Yaskawa INFORM job: DEMO_ROOF_SIDE_0625_3PAINT_38.JBI

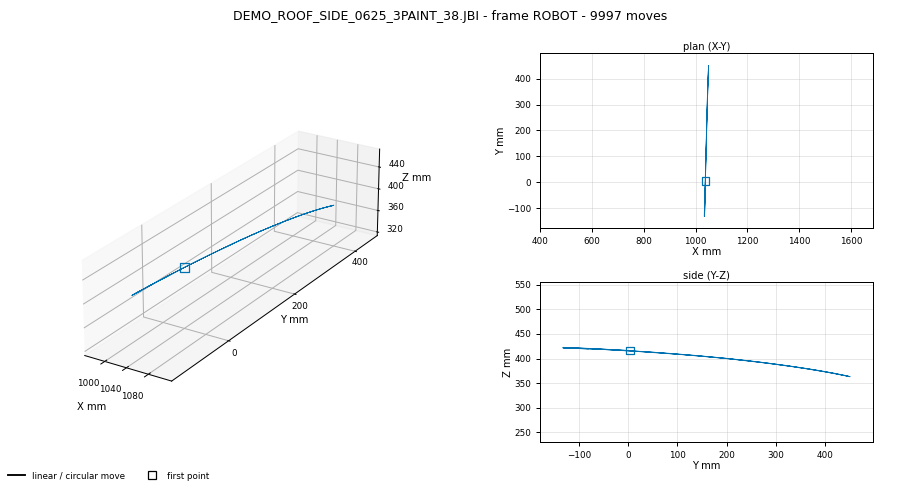
[picture p0: tool path of DEMO_ROOF_SIDE_0625_3PAINT_38.JBI in frame ROBOT, 9997 of 9997 moves have a stored position in this frame; points joined in program order, loops and branches not executed]
/JOB
//NAME DEMO_ROOF_SIDE_0625_3PAINT38
//POS
///NPOS 9997,0,0,0,0,0
///TOOL 0
///USER 0
///POSTYPE ROBOT
///RECTAN
///RCONF 1,0,0,0,0,0,0,0,0,0,0,0,0,0,0,0,0,0,0,0,0,0,0,0
C00000=1038.595,4.241,416.318,169.157,38.319,157.198
C00001=1038.590,3.992,416.332,169.155,38.320,157.198
C00002=1038.583,3.742,416.347,169.153,38.319,157.198
C00003=1038.577,3.493,416.362,169.151,38.318,157.198
C00004=1038.570,3.243,416.378,169.149,38.318,157.198
C00005=1038.564,2.994,416.393,169.147,38.318,157.198
C00006=1038.557,2.744,416.408,169.145,38.317,157.197
C00007=1038.552,2.495,416.422,169.142,38.317,157.197
C00008=1038.545,2.246,416.437,169.140,38.317,157.197
C00009=1038.539,1.996,416.452,169.138,38.316,157.197
C00010=1038.532,1.746,416.467,169.136,38.316,157.197
C00011=1038.526,1.497,416.482,169.134,38.315,157.197
C00012=1038.519,1.248,416.498,169.132,38.315,157.197
C00013=1038.514,0.999,416.513,169.130,38.315,157.197
C00014=1038.507,0.749,416.527,169.128,38.314,157.197
C00015=1038.501,0.499,416.542,169.125,38.314,157.196
C00016=1038.495,0.249,416.558,169.123,38.314,157.196
C00017=1038.489,-0.000,416.573,169.121,38.313,157.196
C00018=1038.483,-0.249,416.587,169.119,38.313,157.196
C00019=1038.477,-0.499,416.602,169.116,38.313,157.196
C00020=1038.470,-0.749,416.617,169.114,38.312,157.196
C00021=1038.464,-0.998,416.632,169.112,38.312,157.196
C00022=1038.458,-1.247,416.647,169.110,38.311,157.196
C00023=1038.452,-1.497,416.662,169.108,38.311,157.196
C00024=1038.445,-1.747,416.677,169.106,38.311,157.196
C00025=1038.439,-1.996,416.692,169.104,38.310,157.195
C00026=1038.433,-2.245,416.706,169.102,38.310,157.195
C00027=1038.427,-2.495,416.721,169.100,38.310,157.195
C00028=1038.420,-2.744,416.736,169.098,38.309,157.195
C00029=1038.414,-2.994,416.751,169.096,38.309,157.195
C00030=1038.407,-3.278,416.767,169.092,38.308,157.195
C00031=1038.400,-3.560,416.785,169.090,38.308,157.195
C00032=1038.393,-3.844,416.802,169.087,38.308,157.195
C00033=1038.385,-4.127,416.817,169.085,38.307,157.194
C00034=1038.379,-4.377,416.832,169.083,38.307,157.194
C00035=1038.373,-4.627,416.847,169.081,38.307,157.194
C00036=1038.366,-4.876,416.862,169.079,38.307,157.194
C00037=1038.360,-5.125,416.876,169.076,38.306,157.194
C00038=1038.354,-5.375,416.890,169.074,38.306,157.194
C00039=1038.347,-5.625,416.905,169.072,38.306,157.194
C00040=1038.340,-5.874,416.920,169.070,38.306,157.194
C00041=1038.334,-6.123,416.934,169.068,38.305,157.194
C00042=1038.328,-6.373,416.949,169.066,38.306,157.194
C00043=1038.321,-6.623,416.963,169.064,38.305,157.194
C00044=1038.315,-6.873,416.978,169.061,38.304,157.193
C00045=1038.309,-7.122,416.992,169.058,38.305,157.193
C00046=1038.303,-7.371,417.007,169.056,38.304,157.193
C00047=1038.296,-7.621,417.021,169.054,38.304,157.193
C00048=1038.290,-7.870,417.035,169.052,38.304,157.193
C00049=1038.284,-8.120,417.050,169.050,38.304,157.193
C00050=1038.277,-8.369,417.065,169.048,38.303,157.193
C00051=1038.271,-8.619,417.079,169.046,38.303,157.193
C00052=1038.265,-8.868,417.094,169.043,38.303,157.193
C00053=1038.258,-9.118,417.108,169.041,38.303,157.193
C00054=1038.252,-9.367,417.123,169.039,38.302,157.193
C00055=1038.246,-9.617,417.137,169.037,38.302,157.192
C00056=1038.239,-9.866,417.151,169.035,38.302,157.192
C00057=1038.233,-10.115,417.166,169.033,38.301,157.192
C00058=1038.227,-10.365,417.180,169.030,38.301,157.192
C00059=1038.220,-10.615,417.194,169.027,38.301,157.192
C00060=1038.214,-10.864,417.209,169.025,38.301,157.192
C00061=1038.208,-11.114,417.223,169.023,38.300,157.192
C00062=1038.201,-11.363,417.237,169.021,38.300,157.192
C00063=1038.195,-11.613,417.251,169.019,38.300,157.192
C00064=1038.189,-11.863,417.266,169.017,38.299,157.192
C00065=1038.182,-12.111,417.280,169.015,38.299,157.192
C00066=1038.176,-12.362,417.294,169.012,38.299,157.191
C00067=1038.170,-12.611,417.309,169.010,38.299,157.191
C00068=1038.163,-12.860,417.323,169.008,38.298,157.191
C00069=1038.157,-13.110,417.338,169.006,38.299,157.191
C00070=1038.151,-13.359,417.352,169.004,38.298,157.191
C00071=1038.145,-13.609,417.366,169.002,38.298,157.191
C00072=1038.139,-13.858,417.380,168.998,38.298,157.191
C00073=1038.132,-14.108,417.394,168.996,38.298,157.191
C00074=1038.126,-14.358,417.409,168.994,38.297,157.191
C00075=1038.120,-14.607,417.423,168.992,38.297,157.191
C00076=1038.113,-14.857,417.437,168.990,38.297,157.191
C00077=1038.107,-15.105,417.452,168.988,38.296,157.190
C00078=1038.101,-15.356,417.466,168.985,38.296,157.190
C00079=1038.095,-15.605,417.479,168.983,38.296,157.190
C00080=1038.088,-15.854,417.494,168.981,38.296,157.190
C00081=1038.082,-16.105,417.508,168.979,38.296,157.190
C00082=1038.075,-16.353,417.522,168.977,38.295,157.190
C00083=1038.069,-16.604,417.536,168.974,38.295,157.190
C00084=1038.063,-16.852,417.550,168.972,38.295,157.190
C00085=1038.056,-17.102,417.564,168.970,38.295,157.190
C00086=1038.050,-17.352,417.578,168.968,38.294,157.190
C00087=1038.043,-17.601,417.592,168.966,38.295,157.190
C00088=1038.037,-17.851,417.606,168.963,38.295,157.190
C00089=1038.031,-18.100,417.620,168.960,38.294,157.190
C00090=1038.024,-18.350,417.634,168.958,38.294,157.190
C00091=1038.018,-18.600,417.648,168.956,38.294,157.189
C00092=1038.011,-18.849,417.662,168.954,38.294,157.189
C00093=1038.005,-19.098,417.675,168.951,38.294,157.189
C00094=1037.998,-19.380,417.692,168.949,38.293,157.189
C00095=1037.992,-19.662,417.707,168.946,38.293,157.189
C00096=1037.984,-19.944,417.723,168.944,38.293,157.189
C00097=1037.977,-20.226,417.738,168.941,38.293,157.189
C00098=1037.970,-20.475,417.752,168.939,38.292,157.189
C00099=1037.964,-20.725,417.766,168.937,38.293,157.189
C00100=1037.958,-20.975,417.780,168.935,38.293,157.189
C00101=1037.951,-21.224,417.794,168.932,38.292,157.189
C00102=1037.945,-21.473,417.808,168.930,38.292,157.189
C00103=1037.939,-21.723,417.822,168.928,38.292,157.188
C00104=1037.932,-21.973,417.835,168.926,38.292,157.188
C00105=1037.926,-22.223,417.849,168.923,38.291,157.188
C00106=1037.920,-22.472,417.863,168.920,38.291,157.188
C00107=1037.914,-22.721,417.877,168.918,38.291,157.188
C00108=1037.908,-22.971,417.891,168.916,38.291,157.188
C00109=1037.901,-23.220,417.904,168.914,38.291,157.188
C00110=1037.894,-23.470,417.918,168.911,38.290,157.188
C00111=1037.889,-23.719,417.932,168.909,38.291,157.188
C00112=1037.882,-23.969,417.946,168.907,38.291,157.188
C00113=1037.876,-24.219,417.959,168.905,38.290,157.188
C00114=1037.870,-24.468,417.973,168.903,38.290,157.188
C00115=1037.863,-24.717,417.987,168.900,38.290,157.188
C00116=1037.857,-24.967,418.001,168.898,38.290,157.188
C00117=1037.851,-25.217,418.015,168.896,38.290,157.188
C00118=1037.845,-25.466,418.028,168.894,38.289,157.187
C00119=1037.838,-25.716,418.041,168.891,38.289,157.187
C00120=1037.832,-25.966,418.056,168.889,38.289,157.187
C00121=1037.826,-26.215,418.069,168.887,38.289,157.187
C00122=1037.820,-26.464,418.082,168.885,38.288,157.187
C00123=1037.813,-26.714,418.097,168.881,38.289,157.187
C00124=1037.807,-26.963,418.110,168.879,38.289,157.187
C00125=1037.800,-27.213,418.124,168.877,38.288,157.187
C00126=1037.794,-27.462,418.137,168.875,38.288,157.187
C00127=1037.789,-27.712,418.151,168.872,38.288,157.187
C00128=1037.782,-27.962,418.165,168.870,38.288,157.187
C00129=1037.776,-28.211,418.178,168.868,38.288,157.187
C00130=1037.769,-28.461,418.191,168.865,38.288,157.187
C00131=1037.763,-28.711,418.205,168.863,38.288,157.187
C00132=1037.756,-28.960,418.218,168.861,38.288,157.187
C00133=1037.750,-29.210,418.232,168.859,38.288,157.186
C00134=1037.743,-29.459,418.245,168.856,38.288,157.186
C00135=1037.737,-29.708,418.258,168.854,38.288,157.186
C00136=1037.731,-29.959,418.271,168.852,38.287,157.186
C00137=1037.725,-30.208,418.285,168.849,38.287,157.186
C00138=1037.718,-30.457,418.298,168.847,38.288,157.186
C00139=1037.712,-30.708,418.312,168.845,38.288,157.186
C00140=1037.706,-30.957,418.325,168.843,38.287,157.186
C00141=1037.700,-31.206,418.339,168.840,38.287,157.186
C00142=1037.693,-31.456,418.352,168.838,38.287,157.186
C00143=1037.687,-31.705,418.366,168.836,38.287,157.186
C00144=1037.681,-31.955,418.379,168.833,38.287,157.186
C00145=1037.674,-32.204,418.392,168.831,38.287,157.186
C00146=1037.668,-32.455,418.405,168.829,38.287,157.186
C00147=1037.662,-32.704,418.418,168.826,38.287,157.186
C00148=1037.655,-32.953,418.432,168.823,38.287,157.185
C00149=1037.649,-33.203,418.445,168.821,38.287,157.185
C00150=1037.642,-33.452,418.458,168.819,38.287,157.185
C00151=1037.636,-33.702,418.472,168.816,38.287,157.185
C00152=1037.630,-33.951,418.485,168.814,38.286,157.185
C00153=1037.623,-34.201,418.498,168.812,38.287,157.185
C00154=1037.617,-34.451,418.511,168.809,38.287,157.185
C00155=1037.611,-34.700,418.524,168.807,38.287,157.185
C00156=1037.605,-34.949,418.538,168.805,38.286,157.185
C00157=1037.598,-35.200,418.551,168.802,38.286,157.185
C00158=1037.592,-35.480,418.566,168.800,38.286,157.185
C00159=1037.585,-35.762,418.580,168.797,38.287,157.185
C00160=1037.578,-36.043,418.596,168.795,38.286,157.185
C00161=1037.571,-36.323,418.610,168.792,38.286,157.185
C00162=1037.564,-36.573,418.624,168.790,38.286,157.185
C00163=1037.558,-36.823,418.637,168.787,38.286,157.185
C00164=1037.552,-37.073,418.650,168.785,38.286,157.185
C00165=1037.546,-37.322,418.663,168.783,38.286,157.185
C00166=1037.540,-37.571,418.676,168.780,38.286,157.184
C00167=1037.533,-37.822,418.689,168.778,38.286,157.184
C00168=1037.527,-38.071,418.702,168.776,38.286,157.184
C00169=1037.521,-38.320,418.716,168.773,38.286,157.184
C00170=1037.515,-38.570,418.728,168.771,38.286,157.184
C00171=1037.508,-38.819,418.742,168.769,38.286,157.184
C00172=1037.502,-39.069,418.755,168.766,38.286,157.184
C00173=1037.496,-39.319,418.768,168.763,38.286,157.184
C00174=1037.490,-39.568,418.781,168.761,38.286,157.184
C00175=1037.483,-39.818,418.793,168.758,38.286,157.184
C00176=1037.477,-40.067,418.806,168.756,38.286,157.184
C00177=1037.470,-40.317,418.820,168.754,38.286,157.184
C00178=1037.465,-40.566,418.832,168.751,38.286,157.184
C00179=1037.458,-40.816,418.846,168.749,38.286,157.184
C00180=1037.451,-41.066,418.858,168.746,38.286,157.184
C00181=1037.445,-41.315,418.871,168.744,38.286,157.184
C00182=1037.439,-41.565,418.883,168.742,38.286,157.184
C00183=1037.433,-41.814,418.897,168.739,38.287,157.184
C00184=1037.426,-42.064,418.909,168.737,38.286,157.184
C00185=1037.420,-42.313,418.922,168.735,38.286,157.184
C00186=1037.413,-42.564,418.935,168.732,38.286,157.184
C00187=1037.407,-42.813,418.948,168.730,38.286,157.184
C00188=1037.401,-43.063,418.960,168.727,38.287,157.184
C00189=1037.394,-43.312,418.973,168.725,38.287,157.184
C00190=1037.388,-43.562,418.986,168.723,38.287,157.183
C00191=1037.382,-43.811,418.999,168.720,38.287,157.183
C00192=1037.376,-44.061,419.012,168.718,38.287,157.183
C00193=1037.370,-44.310,419.024,168.716,38.287,157.183
C00194=1037.363,-44.560,419.037,168.713,38.287,157.183
C00195=1037.358,-44.810,419.050,168.711,38.287,157.183
C00196=1037.351,-45.059,419.063,168.708,38.287,157.183
C00197=1037.345,-45.308,419.075,168.706,38.287,157.183
C00198=1037.338,-45.559,419.088,168.704,38.287,157.183
C00199=1037.332,-45.808,419.101,168.701,38.287,157.183
C00200=1037.325,-46.058,419.113,168.699,38.287,157.183
C00201=1037.319,-46.307,419.126,168.696,38.287,157.183
C00202=1037.313,-46.557,419.139,168.694,38.287,157.183
C00203=1037.307,-46.807,419.151,168.692,38.288,157.183
C00204=1037.300,-47.056,419.164,168.689,38.288,157.183
C00205=1037.294,-47.306,419.177,168.687,38.288,157.183
C00206=1037.288,-47.556,419.189,168.684,38.288,157.183
C00207=1037.282,-47.805,419.202,168.682,38.288,157.183
C00208=1037.276,-48.054,419.214,168.680,38.288,157.183
C00209=1037.270,-48.304,419.227,168.677,38.288,157.183
C00210=1037.264,-48.554,419.239,168.675,38.288,157.183
C00211=1037.257,-48.803,419.252,168.673,38.288,157.183
C00212=1037.251,-49.053,419.265,168.670,38.288,157.183
C00213=1037.245,-49.303,419.277,168.668,38.288,157.183
C00214=1037.239,-49.552,419.290,168.665,38.288,157.183
C00215=1037.232,-49.802,419.302,168.663,38.288,157.183
C00216=1037.227,-50.051,419.315,168.659,38.288,157.183
C00217=1037.221,-50.301,419.327,168.657,38.288,157.182
C00218=1037.214,-50.550,419.339,168.655,38.289,157.182
C00219=1037.208,-50.800,419.352,168.652,38.289,157.182
C00220=1037.201,-51.049,419.364,168.650,38.289,157.182
C00221=1037.196,-51.299,419.377,168.648,38.290,157.182
C00222=1037.188,-51.581,419.390,168.646,38.290,157.182
C00223=1037.180,-51.862,419.404,168.642,38.290,157.182
C00224=1037.173,-52.144,419.418,168.639,38.290,157.182
C00225=1037.166,-52.426,419.433,168.636,38.290,157.182
C00226=1037.160,-52.675,419.444,168.635,38.291,157.182
C00227=1037.153,-52.924,419.456,168.632,38.291,157.182
C00228=1037.147,-53.174,419.469,168.630,38.291,157.182
C00229=1037.141,-53.424,419.481,168.626,38.291,157.182
C00230=1037.134,-53.673,419.493,168.624,38.291,157.182
C00231=1037.128,-53.923,419.505,168.621,38.291,157.182
C00232=1037.122,-54.173,419.517,168.620,38.292,157.182
C00233=1037.115,-54.422,419.529,168.617,38.292,157.182
C00234=1037.109,-54.672,419.542,168.615,38.292,157.182
C00235=1037.102,-54.922,419.554,168.612,38.293,157.182
C00236=1037.096,-55.172,419.566,168.609,38.293,157.182
C00237=1037.090,-55.421,419.578,168.607,38.293,157.182
C00238=1037.083,-55.671,419.590,168.605,38.294,157.182
C00239=1037.077,-55.921,419.603,168.602,38.294,157.182
C00240=1037.071,-56.170,419.615,168.600,38.294,157.182
C00241=1037.065,-56.419,419.626,168.597,38.294,157.182
C00242=1037.059,-56.669,419.639,168.595,38.295,157.182
C00243=1037.052,-56.919,419.651,168.592,38.295,157.182
C00244=1037.045,-57.168,419.663,168.590,38.295,157.182
C00245=1037.039,-57.418,419.675,168.588,38.295,157.182
C00246=1037.033,-57.668,419.687,168.585,38.295,157.182
C00247=1037.026,-57.918,419.698,168.583,38.296,157.182
C00248=1037.020,-58.167,419.710,168.580,38.296,157.182
C00249=1037.014,-58.416,419.723,168.578,38.296,157.182
C00250=1037.008,-58.666,419.735,168.575,38.296,157.182
C00251=1037.001,-58.916,419.746,168.573,38.296,157.182
C00252=1036.995,-59.166,419.759,168.570,38.297,157.182
C00253=1036.989,-59.415,419.771,168.568,38.297,157.182
C00254=1036.983,-59.664,419.783,168.565,38.297,157.182
C00255=1036.977,-59.914,419.794,168.563,38.297,157.182
C00256=1036.970,-60.164,419.806,168.560,38.298,157.182
C00257=1036.964,-60.414,419.818,168.558,38.298,157.182
C00258=1036.958,-60.663,419.831,168.555,38.298,157.182
C00259=1036.952,-60.912,419.843,168.553,38.299,157.182
C00260=1036.945,-61.163,419.854,168.550,38.299,157.182
C00261=1036.939,-61.412,419.866,168.548,38.299,157.182
C00262=1036.933,-61.662,419.878,168.545,38.300,157.182
C00263=1036.926,-61.912,419.890,168.543,38.300,157.182
C00264=1036.920,-62.160,419.902,168.540,38.300,157.182
C00265=1036.915,-62.411,419.914,168.538,38.300,157.182
C00266=1036.908,-62.661,419.926,168.535,38.301,157.182
C00267=1036.901,-62.910,419.938,168.533,38.301,157.182
C00268=1036.895,-63.159,419.949,168.530,38.301,157.182
C00269=1036.890,-63.409,419.961,168.527,38.301,157.182
C00270=1036.883,-63.659,419.973,168.525,38.302,157.182
C00271=1036.877,-63.908,419.985,168.522,38.302,157.182
C00272=1036.871,-64.158,419.996,168.520,38.302,157.182
C00273=1036.865,-64.408,420.008,168.517,38.302,157.182
C00274=1036.858,-64.658,420.020,168.515,38.303,157.182
C00275=1036.852,-64.907,420.031,168.512,38.303,157.182
C00276=1036.846,-65.157,420.044,168.510,38.303,157.182
C00277=1036.840,-65.407,420.056,168.507,38.303,157.182
C00278=1036.834,-65.656,420.067,168.505,38.303,157.182
C00279=1036.827,-65.906,420.079,168.502,38.304,157.182
C00280=1036.821,-66.155,420.091,168.500,38.304,157.182
C00281=1036.816,-66.405,420.102,168.497,38.304,157.182
C00282=1036.809,-66.655,420.114,168.495,38.305,157.182
C00283=1036.802,-66.904,420.126,168.492,38.305,157.182
C00284=1036.797,-67.154,420.137,168.490,38.305,157.182
C00285=1036.791,-67.403,420.149,168.487,38.306,157.182
C00286=1036.784,-67.686,420.162,168.484,38.306,157.182
C00287=1036.777,-67.969,420.175,168.481,38.307,157.182
C00288=1036.770,-68.252,420.189,168.479,38.307,157.182
C00289=1036.763,-68.535,420.202,168.476,38.307,157.182
C00290=1036.757,-68.784,420.214,168.473,38.308,157.182
C00291=1036.751,-69.034,420.225,168.471,38.308,157.182
C00292=1036.745,-69.284,420.237,168.468,38.308,157.182
C00293=1036.739,-69.533,420.248,168.466,38.308,157.182
C00294=1036.733,-69.783,420.260,168.463,38.309,157.182
C00295=1036.726,-70.033,420.271,168.461,38.309,157.182
C00296=1036.720,-70.282,420.283,168.458,38.309,157.182
C00297=1036.715,-70.532,420.295,168.455,38.309,157.182
C00298=1036.708,-70.781,420.306,168.453,38.310,157.182
C00299=1036.702,-71.032,420.317,168.450,38.310,157.182
C00300=1036.696,-71.280,420.329,168.448,38.310,157.182
C00301=1036.690,-71.531,420.341,168.445,38.311,157.182
C00302=1036.684,-71.780,420.352,168.443,38.311,157.182
C00303=1036.678,-72.030,420.364,168.440,38.311,157.182
C00304=1036.672,-72.279,420.375,168.438,38.311,157.182
C00305=1036.666,-72.529,420.387,168.435,38.312,157.182
C00306=1036.661,-72.779,420.398,168.433,38.312,157.182
C00307=1036.654,-73.028,420.410,168.430,38.312,157.182
C00308=1036.648,-73.278,420.421,168.428,38.312,157.182
C00309=1036.642,-73.528,420.432,168.425,38.313,157.182
C00310=1036.635,-73.778,420.444,168.422,38.313,157.182
C00311=1036.630,-74.027,420.455,168.420,38.313,157.182
C00312=1036.624,-74.278,420.467,168.417,38.314,157.182
C00313=1036.617,-74.526,420.478,168.415,38.314,157.182
C00314=1036.611,-74.776,420.489,168.412,38.315,157.182
C00315=1036.605,-75.026,420.500,168.410,38.315,157.182
C00316=1036.598,-75.275,420.512,168.407,38.316,157.182
C00317=1036.593,-75.525,420.523,168.404,38.316,157.182
C00318=1036.586,-75.775,420.534,168.402,38.317,157.182
C00319=1036.581,-76.025,420.545,168.399,38.317,157.182
C00320=1036.574,-76.274,420.557,168.397,38.318,157.182
C00321=1036.568,-76.524,420.568,168.394,38.318,157.182
C00322=1036.562,-76.774,420.579,168.392,38.319,157.182
C00323=1036.556,-77.023,420.590,168.390,38.319,157.182
C00324=1036.550,-77.274,420.601,168.387,38.320,157.182
C00325=1036.544,-77.522,420.613,168.385,38.320,157.182
C00326=1036.537,-77.773,420.624,168.382,38.320,157.183
C00327=1036.531,-78.022,420.634,168.379,38.321,157.182
C00328=1036.525,-78.271,420.645,168.377,38.321,157.183
C00329=1036.519,-78.521,420.656,168.374,38.321,157.183
C00330=1036.513,-78.771,420.667,168.372,38.322,157.183
C00331=1036.507,-79.021,420.679,168.369,38.322,157.183
C00332=1036.501,-79.270,420.690,168.366,38.323,157.183
C00333=1036.494,-79.520,420.701,168.364,38.323,157.183
C00334=1036.489,-79.770,420.712,168.361,38.324,157.183
C00335=1036.483,-80.019,420.723,168.359,38.324,157.183
C00336=1036.476,-80.269,420.734,168.356,38.325,157.183
C00337=1036.470,-80.519,420.744,168.353,38.325,157.183
C00338=1036.464,-80.769,420.756,168.351,38.326,157.183
C00339=1036.457,-81.018,420.766,168.348,38.327,157.183
C00340=1036.451,-81.268,420.777,168.345,38.327,157.183
C00341=1036.445,-81.518,420.788,168.343,38.328,157.183
C00342=1036.438,-81.767,420.799,168.340,38.328,157.183
C00343=1036.432,-82.017,420.810,168.337,38.329,157.183
C00344=1036.427,-82.266,420.821,168.335,38.329,157.183
C00345=1036.420,-82.516,420.831,168.333,38.330,157.183
C00346=1036.414,-82.766,420.842,168.330,38.331,157.183
C00347=1036.408,-83.016,420.853,168.328,38.331,157.183
C00348=1036.401,-83.265,420.864,168.325,38.332,157.183
C00349=1036.395,-83.515,420.874,168.322,38.333,157.183
C00350=1036.388,-83.800,420.887,168.319,38.333,157.183
C00351=1036.381,-84.085,420.899,168.316,38.334,157.183
C00352=1036.374,-84.370,420.911,168.313,38.334,157.184
C00353=1036.367,-84.655,420.923,168.310,38.335,157.184
C00354=1036.361,-84.905,420.934,168.308,38.336,157.184
C00355=1036.354,-85.154,420.944,168.305,38.336,157.184
C00356=1036.349,-85.404,420.955,168.302,38.337,157.184
C00357=1036.342,-85.654,420.967,168.300,38.338,157.184
C00358=1036.336,-85.903,420.977,168.297,38.338,157.184
C00359=1036.330,-86.152,420.988,168.294,38.339,157.184
C00360=1036.323,-86.402,420.998,168.292,38.339,157.184
C00361=1036.318,-86.652,421.009,168.289,38.340,157.184
C00362=1036.312,-86.902,421.019,168.286,38.340,157.184
C00363=1036.305,-87.152,421.030,168.285,38.341,157.184
C00364=1036.299,-87.401,421.041,168.282,38.342,157.184
C00365=1036.293,-87.651,421.052,168.279,38.343,157.184
C00366=1036.287,-87.901,421.061,168.277,38.343,157.184
C00367=1036.281,-88.151,421.073,168.274,38.343,157.184
C00368=1036.274,-88.400,421.083,168.271,38.344,157.184
C00369=1036.269,-88.649,421.094,168.268,38.345,157.184
C00370=1036.263,-88.900,421.104,168.266,38.345,157.184
C00371=1036.256,-89.149,421.115,168.263,38.346,157.185
C00372=1036.250,-89.399,421.126,168.260,38.347,157.185
C00373=1036.244,-89.648,421.136,168.258,38.348,157.185
C00374=1036.238,-89.899,421.146,168.255,38.348,157.185
C00375=1036.232,-90.148,421.157,168.252,38.349,157.185
C00376=1036.226,-90.398,421.167,168.250,38.349,157.185
C00377=1036.220,-90.648,421.178,168.247,38.350,157.185
C00378=1036.214,-90.897,421.188,168.244,38.350,157.185
C00379=1036.207,-91.147,421.199,168.242,38.351,157.185
C00380=1036.201,-91.396,421.209,168.240,38.352,157.185
C00381=1036.195,-91.646,421.220,168.237,38.353,157.185
C00382=1036.190,-91.896,421.230,168.235,38.353,157.185
C00383=1036.184,-92.146,421.240,168.232,38.353,157.185
C00384=1036.178,-92.395,421.251,168.229,38.354,157.185
C00385=1036.171,-92.645,421.262,168.227,38.355,157.185
C00386=1036.165,-92.895,421.272,168.224,38.355,157.185
C00387=1036.160,-93.145,421.283,168.221,38.356,157.185
C00388=1036.153,-93.394,421.293,168.219,38.357,157.185
C00389=1036.148,-93.644,421.303,168.216,38.358,157.186
C00390=1036.141,-93.893,421.313,168.213,38.358,157.186
C00391=1036.135,-94.144,421.324,168.211,38.358,157.186
C00392=1036.129,-94.393,421.334,168.208,38.359,157.186
C00393=1036.123,-94.643,421.344,168.205,38.360,157.186
C00394=1036.117,-94.892,421.355,168.202,38.361,157.186
C00395=1036.111,-95.142,421.365,168.200,38.361,157.186
C00396=1036.106,-95.392,421.376,168.197,38.362,157.186
C00397=1036.099,-95.641,421.386,168.195,38.363,157.186
C00398=1036.094,-95.891,421.396,168.193,38.363,157.186
C00399=1036.087,-96.140,421.406,168.190,38.364,157.186
C00400=1036.082,-96.390,421.417,168.187,38.364,157.186
C00401=1036.075,-96.640,421.427,168.185,38.365,157.186
C00402=1036.069,-96.890,421.437,168.182,38.366,157.186
C00403=1036.063,-97.140,421.448,168.179,38.367,157.186
C00404=1036.057,-97.390,421.458,168.177,38.367,157.186
C00405=1036.051,-97.640,421.467,168.174,38.368,157.187
C00406=1036.045,-97.889,421.478,168.171,38.369,157.187
C00407=1036.039,-98.139,421.488,168.168,38.370,157.187
C00408=1036.033,-98.388,421.498,168.166,38.371,157.187
C00409=1036.027,-98.638,421.508,168.163,38.371,157.187
C00410=1036.021,-98.888,421.518,168.161,38.372,157.187
C00411=1036.015,-99.137,421.528,168.158,38.373,157.187
C00412=1036.008,-99.387,421.538,168.156,38.374,157.187
C00413=1036.002,-99.638,421.548,168.153,38.375,157.187
C00414=1035.993,-100.042,421.564,168.148,38.376,157.187
C00415=1035.983,-100.445,421.581,168.144,38.377,157.187
C00416=1035.972,-100.849,421.597,168.140,38.378,157.187
C00417=1035.963,-101.253,421.613,168.135,38.379,157.188
C00418=1035.957,-101.503,421.623,168.132,38.380,157.188
C00419=1035.951,-101.753,421.632,168.130,38.381,157.188
C00420=1035.945,-102.002,421.642,168.128,38.382,157.188
C00421=1035.938,-102.252,421.652,168.125,38.383,157.188
C00422=1035.933,-102.502,421.663,168.122,38.383,157.188
C00423=1035.927,-102.752,421.672,168.120,38.384,157.188
C00424=1035.921,-103.001,421.682,168.117,38.385,157.188
C00425=1035.914,-103.251,421.692,168.114,38.386,157.188
C00426=1035.909,-103.501,421.702,168.111,38.387,157.188
C00427=1035.903,-103.750,421.712,168.109,38.387,157.188
C00428=1035.896,-104.000,421.721,168.106,38.388,157.189
C00429=1035.890,-104.250,421.731,168.103,38.389,157.189
C00430=1035.885,-104.500,421.741,168.101,38.391,157.189
C00431=1035.878,-104.749,421.751,168.099,38.391,157.189
C00432=1035.872,-104.999,421.761,168.096,38.392,157.189
C00433=1035.867,-105.248,421.770,168.093,38.393,157.189
C00434=1035.861,-105.498,421.780,168.090,38.394,157.189
C00435=1035.855,-105.748,421.790,168.088,38.394,157.189
C00436=1035.849,-105.998,421.799,168.085,38.395,157.189
C00437=1035.843,-106.248,421.809,168.082,38.396,157.189
C00438=1035.833,-106.631,421.825,168.078,38.398,157.190
C00439=1035.824,-107.013,421.839,168.074,38.399,157.190
C00440=1035.815,-107.396,421.854,168.070,38.400,157.190
C00441=1035.806,-107.778,421.868,168.066,38.402,157.190
C00442=1035.799,-108.027,421.878,168.063,38.402,157.190
C00443=1035.794,-108.278,421.888,168.061,38.403,157.190
C00444=1035.788,-108.527,421.898,168.058,38.405,157.190
C00445=1035.782,-108.777,421.907,168.055,38.405,157.190
C00446=1035.775,-109.027,421.917,168.052,38.406,157.190
C00447=1035.769,-109.277,421.926,168.049,38.407,157.191
C00448=1035.763,-109.527,421.936,168.047,38.408,157.191
C00449=1035.757,-109.776,421.945,168.045,38.409,157.191
C00450=1035.751,-110.025,421.955,168.042,38.410,157.191
C00451=1035.745,-110.276,421.964,168.039,38.411,157.191
C00452=1035.739,-110.526,421.973,168.036,38.412,157.191
C00453=1035.733,-110.775,421.983,168.034,38.413,157.191
C00454=1035.727,-111.025,421.992,168.031,38.414,157.191
C00455=1035.721,-111.275,422.002,168.028,38.415,157.191
C00456=1035.715,-111.524,422.011,168.025,38.416,157.191
C00457=1035.709,-111.774,422.021,168.022,38.417,157.192
C00458=1035.703,-112.024,422.030,168.021,38.418,157.192
C00459=1035.697,-112.274,422.040,168.018,38.419,157.192
C00460=1035.691,-112.523,422.049,168.015,38.419,157.192
C00461=1035.685,-112.773,422.058,168.012,38.421,157.192
C00462=1035.679,-113.023,422.067,168.009,38.422,157.192
C00463=1035.673,-113.273,422.077,168.007,38.423,157.192
C00464=1035.667,-113.522,422.086,168.004,38.423,157.192
C00465=1035.661,-113.772,422.096,168.001,38.425,157.193
C00466=1035.655,-114.021,422.105,167.998,38.426,157.193
C00467=1035.649,-114.272,422.114,167.996,38.426,157.193
C00468=1035.643,-114.522,422.124,167.994,38.427,157.193
C00469=1035.637,-114.771,422.133,167.991,38.429,157.193
C00470=1035.631,-115.020,422.142,167.988,38.430,157.193
C00471=1035.625,-115.271,422.151,167.985,38.430,157.193
C00472=1035.619,-115.521,422.161,167.982,38.432,157.193
C00473=1035.613,-115.770,422.170,167.980,38.433,157.193
C00474=1035.606,-116.056,422.180,167.976,38.434,157.194
C00475=1035.599,-116.343,422.191,167.973,38.435,157.194
C00476=1035.593,-116.629,422.202,167.971,38.436,157.194
C00477=1035.586,-116.916,422.212,167.968,38.437,157.194
C00478=1035.579,-117.166,422.221,167.965,38.439,157.194
C00479=1035.573,-117.416,422.231,167.962,38.440,157.194
C00480=1035.568,-117.666,422.239,167.959,38.440,157.194
C00481=1035.562,-117.915,422.249,167.956,38.442,157.194
C00482=1035.556,-118.165,422.258,167.954,38.443,157.194
C00483=1035.550,-118.415,422.267,167.952,38.444,157.195
C00484=1035.543,-118.664,422.276,167.949,38.445,157.195
C00485=1035.537,-118.914,422.285,167.946,38.446,157.195
C00486=1035.532,-119.164,422.294,167.943,38.447,157.195
C00487=1035.526,-119.414,422.303,167.940,38.448,157.195
C00488=1035.520,-119.664,422.312,167.938,38.449,157.195
C00489=1035.514,-119.913,422.321,167.935,38.450,157.195
C00490=1035.508,-120.163,422.330,167.932,38.452,157.196
C00491=1035.502,-120.413,422.339,167.930,38.453,157.196
C00492=1035.496,-120.662,422.349,167.927,38.454,157.196
C00493=1035.490,-120.913,422.357,167.924,38.455,157.196
C00494=1035.484,-121.162,422.367,167.922,38.456,157.196
C00495=1035.478,-121.412,422.375,167.919,38.457,157.196
C00496=1035.472,-121.662,422.384,167.916,38.458,157.196
C00497=1035.467,-121.911,422.393,167.913,38.459,157.196
C00498=1035.460,-122.161,422.402,167.910,38.460,157.197
C00499=1035.455,-122.412,422.411,167.908,38.462,157.197
C00500=1035.448,-122.660,422.420,167.906,38.463,157.197
C00501=1035.442,-122.911,422.429,167.903,38.464,157.197
C00502=1035.437,-123.160,422.438,167.900,38.465,157.197
C00503=1035.431,-123.410,422.447,167.897,38.466,157.197
C00504=1035.424,-123.660,422.456,167.894,38.467,157.197
C00505=1035.419,-123.909,422.464,167.891,38.469,157.198
C00506=1035.413,-124.160,422.473,167.890,38.469,157.198
C00507=1035.407,-124.409,422.482,167.887,38.471,157.198
C00508=1035.401,-124.659,422.491,167.884,38.472,157.198
C00509=1035.395,-124.908,422.500,167.881,38.473,157.198
C00510=1035.389,-125.159,422.509,167.878,38.475,157.198
C00511=1035.383,-125.409,422.517,167.875,38.475,157.198
C00512=1035.377,-125.658,422.526,167.872,38.477,157.199
C00513=1035.371,-125.908,422.535,167.870,38.478,157.199
C00514=1035.365,-126.158,422.543,167.868,38.479,157.199
C00515=1035.359,-126.407,422.552,167.865,38.481,157.199
C00516=1035.353,-126.657,422.560,167.862,38.482,157.199
C00517=1035.347,-126.907,422.569,167.859,38.483,157.199
C00518=1035.342,-127.156,422.578,167.856,38.484,157.199
C00519=1035.335,-127.406,422.587,167.853,38.485,157.199
C00520=1035.330,-127.656,422.595,167.851,38.487,157.200
C00521=1035.324,-127.906,422.605,167.849,38.488,157.200
C00522=1035.318,-128.156,422.613,167.846,38.488,157.200
C00523=1035.314,-128.405,422.624,167.843,38.489,157.200
C00524=1035.311,-128.654,422.634,167.841,38.489,157.200
C00525=1035.307,-128.904,422.645,167.839,38.488,157.200
C00526=1035.305,-129.155,422.656,167.836,38.487,157.199
C00527=1035.303,-129.404,422.669,167.834,38.485,157.199
C00528=1035.303,-129.654,422.681,167.832,38.483,157.199
C00529=1035.303,-129.904,422.695,167.830,38.480,157.198
C00530=1035.303,-130.155,422.709,167.829,38.478,157.198
C00531=1035.304,-130.404,422.723,167.827,38.474,157.197
C00532=1035.307,-130.654,422.739,167.826,38.471,157.196
C00533=1035.309,-130.903,422.755,167.824,38.466,157.196
C00534=1035.313,-131.154,422.770,167.822,38.461,157.195
C00535=1035.317,-131.404,422.788,167.821,38.456,157.194
C00536=1035.322,-131.655,422.806,167.820,38.451,157.193
C00537=1035.327,-131.904,422.824,167.819,38.444,157.192
C00538=1034.993,-131.929,422.544,167.770,38.661,157.227
C00539=1034.988,-131.679,422.525,167.771,38.667,157.228
C00540=1034.983,-131.429,422.508,167.772,38.673,157.229
C00541=1034.979,-131.179,422.491,167.774,38.678,157.230
C00542=1034.975,-130.928,422.475,167.775,38.683,157.231
C00543=1034.973,-130.678,422.459,167.777,38.687,157.232
C00544=1034.971,-130.429,422.443,167.778,38.691,157.232
C00545=1034.969,-130.179,422.429,167.780,38.695,157.233
C00546=1034.968,-129.929,422.415,167.782,38.697,157.233
C00547=1034.969,-129.679,422.401,167.784,38.700,157.234
C00548=1034.970,-129.429,422.389,167.786,38.702,157.234
C00549=1034.971,-129.180,422.377,167.788,38.704,157.235
C00550=1034.973,-128.929,422.364,167.790,38.705,157.235
C00551=1034.977,-128.679,422.353,167.793,38.706,157.235
C00552=1034.980,-128.430,422.343,167.795,38.705,157.235
C00553=1034.984,-128.180,422.333,167.797,38.705,157.235
C00554=1034.989,-127.930,422.324,167.800,38.704,157.235
C00555=1034.996,-127.681,422.315,167.803,38.704,157.235
C00556=1035.001,-127.431,422.306,167.806,38.702,157.235
C00557=1035.008,-127.181,422.297,167.808,38.701,157.235
C00558=1035.013,-126.932,422.289,167.811,38.700,157.235
C00559=1035.019,-126.681,422.280,167.814,38.698,157.234
C00560=1035.025,-126.433,422.271,167.816,38.697,157.234
C00561=1035.031,-126.182,422.263,167.819,38.696,157.234
C00562=1035.036,-125.932,422.254,167.822,38.694,157.234
C00563=1035.043,-125.682,422.246,167.824,38.693,157.234
C00564=1035.048,-125.433,422.237,167.827,38.692,157.234
C00565=1035.054,-125.183,422.228,167.830,38.691,157.233
C00566=1035.061,-124.934,422.219,167.833,38.690,157.233
C00567=1035.066,-124.684,422.210,167.836,38.688,157.233
C00568=1035.073,-124.434,422.203,167.838,38.687,157.233
C00569=1035.079,-124.184,422.193,167.841,38.686,157.233
C00570=1035.085,-123.934,422.184,167.843,38.684,157.233
C00571=1035.090,-123.684,422.176,167.846,38.684,157.233
C00572=1035.097,-123.435,422.167,167.849,38.682,157.232
C00573=1035.102,-123.185,422.158,167.852,38.681,157.232
C00574=1035.108,-122.935,422.149,167.855,38.680,157.232
C00575=1035.113,-122.686,422.140,167.857,38.679,157.232
C00576=1035.120,-122.436,422.131,167.860,38.677,157.232
C00577=1035.126,-122.186,422.122,167.862,38.677,157.232
C00578=1035.132,-121.937,422.113,167.865,38.675,157.232
C00579=1035.138,-121.686,422.104,167.868,38.674,157.232
C00580=1035.143,-121.437,422.095,167.871,38.673,157.231
C00581=1035.150,-121.187,422.087,167.874,38.671,157.231
C00582=1035.156,-120.937,422.077,167.877,38.670,157.231
C00583=1035.161,-120.687,422.069,167.879,38.669,157.231
C00584=1035.167,-120.438,422.059,167.881,38.668,157.231
C00585=1035.173,-120.187,422.050,167.884,38.667,157.231
C00586=1035.180,-119.938,422.042,167.887,38.666,157.231
C00587=1035.185,-119.688,422.033,167.890,38.665,157.231
C00588=1035.192,-119.438,422.023,167.893,38.664,157.230
C00589=1035.197,-119.189,422.014,167.895,38.663,157.230
C00590=1035.203,-118.939,422.005,167.898,38.661,157.230
C00591=1035.209,-118.689,421.996,167.901,38.660,157.230
C00592=1035.215,-118.439,421.988,167.903,38.659,157.230
C00593=1035.221,-118.190,421.978,167.906,38.658,157.230
C00594=1035.228,-117.940,421.969,167.909,38.657,157.230
C00595=1035.233,-117.690,421.960,167.912,38.656,157.230
C00596=1035.239,-117.440,421.951,167.914,38.654,157.229
C00597=1035.245,-117.191,421.941,167.917,38.653,157.229
C00598=1035.250,-116.941,421.933,167.920,38.653,157.229
C00599=1035.258,-116.655,421.922,167.922,38.651,157.229
C00600=1035.265,-116.368,421.911,167.926,38.650,157.229
C00601=1035.271,-116.081,421.900,167.929,38.649,157.229
C00602=1035.279,-115.795,421.890,167.932,38.647,157.229
C00603=1035.285,-115.545,421.881,167.935,38.646,157.229
C00604=1035.290,-115.296,421.872,167.938,38.645,157.228
C00605=1035.296,-115.046,421.863,167.941,38.644,157.228
C00606=1035.303,-114.796,421.853,167.942,38.643,157.228
C00607=1035.308,-114.546,421.844,167.945,38.642,157.228
C00608=1035.314,-114.296,421.835,167.948,38.641,157.228
C00609=1035.320,-114.047,421.825,167.951,38.640,157.228
C00610=1035.326,-113.797,421.816,167.954,38.639,157.228
C00611=1035.332,-113.547,421.806,167.957,38.638,157.228
C00612=1035.338,-113.297,421.798,167.959,38.637,157.228
C00613=1035.344,-113.048,421.788,167.962,38.636,157.227
C00614=1035.350,-112.798,421.779,167.964,38.635,157.227
C00615=1035.356,-112.548,421.769,167.967,38.634,157.227
C00616=1035.362,-112.298,421.760,167.970,38.632,157.227
C00617=1035.368,-112.049,421.750,167.972,38.632,157.227
C00618=1035.374,-111.799,421.741,167.975,38.631,157.227
C00619=1035.380,-111.549,421.732,167.978,38.630,157.227
C00620=1035.386,-111.299,421.722,167.981,38.628,157.227
C00621=1035.392,-111.049,421.713,167.984,38.628,157.227
C00622=1035.398,-110.800,421.704,167.987,38.627,157.226
C00623=1035.404,-110.550,421.694,167.988,38.625,157.226
C00624=1035.410,-110.301,421.684,167.991,38.624,157.226
C00625=1035.416,-110.051,421.675,167.994,38.624,157.226
C00626=1035.423,-109.801,421.665,167.997,38.623,157.226
C00627=1035.429,-109.551,421.656,168.000,38.621,157.226
C00628=1035.434,-109.302,421.647,168.002,38.621,157.226
C00629=1035.441,-109.052,421.637,168.005,38.620,157.226
C00630=1035.447,-108.802,421.627,168.008,38.619,157.226
C00631=1035.453,-108.553,421.618,168.010,38.617,157.225
C00632=1035.459,-108.303,421.608,168.013,38.617,157.225
C00633=1035.465,-108.053,421.599,168.015,38.616,157.225
C00634=1035.471,-107.803,421.589,168.018,38.615,157.225
C00635=1035.477,-107.553,421.579,168.021,38.613,157.225
C00636=1035.483,-107.303,421.569,168.024,38.613,157.225
C00637=1035.489,-107.054,421.560,168.027,38.612,157.225
C00638=1035.495,-106.804,421.551,168.029,38.611,157.225
C00639=1035.501,-106.555,421.541,168.032,38.610,157.225
C00640=1035.507,-106.305,421.532,168.034,38.609,157.225
C00641=1035.513,-106.055,421.521,168.037,38.608,157.224
C00642=1035.519,-105.805,421.512,168.040,38.607,157.224
C00643=1035.525,-105.555,421.502,168.042,38.606,157.224
C00644=1035.531,-105.305,421.493,168.045,38.605,157.224
C00645=1035.537,-105.056,421.483,168.048,38.605,157.224
C00646=1035.543,-104.806,421.472,168.051,38.604,157.224
C00647=1035.549,-104.556,421.463,168.053,38.603,157.224
C00648=1035.555,-104.306,421.453,168.056,38.602,157.224
C00649=1035.561,-104.057,421.444,168.059,38.601,157.224
C00650=1035.566,-103.807,421.434,168.062,38.600,157.224
C00651=1035.572,-103.557,421.424,168.064,38.599,157.224
C00652=1035.579,-103.308,421.414,168.066,38.598,157.223
C00653=1035.585,-103.059,421.404,168.069,38.597,157.223
C00654=1035.591,-102.808,421.394,168.072,38.597,157.223
C00655=1035.597,-102.559,421.385,168.075,38.596,157.223
C00656=1035.603,-102.309,421.375,168.077,38.595,157.223
C00657=1035.609,-102.060,421.365,168.080,38.594,157.223
C00658=1035.615,-101.810,421.355,168.083,38.593,157.223
C00659=1035.621,-101.560,421.345,168.086,38.592,157.223
C00660=1035.627,-101.310,421.335,168.089,38.591,157.223
C00661=1035.633,-101.060,421.325,168.090,38.590,157.223
C00662=1035.639,-100.811,421.315,168.093,38.589,157.223
C00663=1035.646,-100.523,421.304,168.096,38.589,157.223
C00664=1035.654,-100.236,421.292,168.099,38.588,157.222
C00665=1035.660,-99.948,421.281,168.103,38.587,157.222
C00666=1035.667,-99.662,421.269,168.106,38.585,157.222
C00667=1035.673,-99.413,421.260,168.109,38.585,157.222
C00668=1035.679,-99.162,421.249,168.111,38.584,157.222
C00669=1035.686,-98.913,421.239,168.114,38.583,157.222
C00670=1035.692,-98.663,421.229,168.117,38.582,157.222
C00671=1035.698,-98.413,421.219,168.119,38.581,157.222
C00672=1035.704,-98.163,421.209,168.121,38.581,157.222
C00673=1035.710,-97.914,421.199,168.124,38.580,157.222
C00674=1035.716,-97.664,421.190,168.127,38.579,157.222
C00675=1035.722,-97.414,421.179,168.130,38.578,157.222
C00676=1035.728,-97.165,421.169,168.132,38.577,157.221
C00677=1035.734,-96.915,421.158,168.135,38.577,157.221
C00678=1035.739,-96.665,421.148,168.138,38.576,157.221
C00679=1035.746,-96.416,421.138,168.140,38.576,157.221
C00680=1035.751,-96.166,421.128,168.143,38.575,157.221
C00681=1035.758,-95.916,421.117,168.146,38.574,157.221
C00682=1035.764,-95.666,421.107,168.149,38.573,157.221
C00683=1035.770,-95.417,421.097,168.151,38.572,157.221
C00684=1035.776,-95.166,421.086,168.153,38.572,157.221
C00685=1035.782,-94.917,421.076,168.156,38.571,157.221
C00686=1035.788,-94.667,421.066,168.158,38.571,157.221
C00687=1035.794,-94.418,421.056,168.161,38.570,157.221
C00688=1035.800,-94.168,421.045,168.164,38.569,157.221
C00689=1035.805,-93.918,421.035,168.167,38.568,157.221
C00690=1035.812,-93.668,421.025,168.169,38.567,157.221
C00691=1035.818,-93.418,421.014,168.172,38.567,157.221
C00692=1035.824,-93.169,421.004,168.175,38.566,157.221
C00693=1035.830,-92.919,420.993,168.177,38.566,157.220
C00694=1035.836,-92.670,420.983,168.180,38.565,157.220
C00695=1035.842,-92.420,420.973,168.183,38.564,157.220
C00696=1035.847,-92.170,420.962,168.185,38.563,157.220
C00697=1035.855,-91.920,420.951,168.188,38.563,157.220
C00698=1035.860,-91.670,420.941,168.191,38.562,157.220
C00699=1035.866,-91.421,420.931,168.193,38.561,157.220
C00700=1035.872,-91.172,420.920,168.195,38.561,157.220
C00701=1035.878,-90.922,420.910,168.198,38.560,157.220
C00702=1035.885,-90.672,420.899,168.201,38.560,157.220
C00703=1035.890,-90.438,420.890,168.203,38.559,157.220
C00704=1035.896,-90.205,420.879,168.206,38.558,157.220
C00705=1035.902,-89.972,420.870,168.208,38.557,157.220
C00706=1035.908,-89.739,420.860,168.211,38.557,157.220
C00707=1035.913,-89.506,420.850,168.213,38.556,157.220
C00708=1035.919,-89.272,420.840,168.216,38.556,157.220
C00709=1035.924,-89.039,420.830,168.218,38.555,157.220
C00710=1035.930,-88.806,420.821,168.221,38.555,157.220
C00711=1035.936,-88.556,420.810,168.224,38.554,157.219
C00712=1035.942,-88.307,420.800,168.226,38.553,157.219
C00713=1035.948,-88.058,420.789,168.229,38.552,157.219
C00714=1035.954,-87.807,420.779,168.231,38.551,157.219
C00715=1035.961,-87.558,420.768,168.234,38.551,157.219
C00716=1035.966,-87.308,420.757,168.236,38.550,157.219
C00717=1035.973,-87.058,420.746,168.239,38.550,157.219
C00718=1035.979,-86.809,420.736,168.241,38.549,157.219
C00719=1035.985,-86.559,420.726,168.244,38.548,157.219
C00720=1035.991,-86.309,420.715,168.247,38.548,157.219
C00721=1035.997,-86.059,420.704,168.249,38.547,157.219
C00722=1036.003,-85.810,420.693,168.252,38.546,157.219
C00723=1036.010,-85.561,420.683,168.255,38.545,157.219
C00724=1036.016,-85.310,420.672,168.257,38.545,157.219
C00725=1036.022,-85.061,420.661,168.260,38.545,157.219
C00726=1036.028,-84.811,420.651,168.263,38.544,157.219
C00727=1036.036,-84.493,420.637,168.266,38.543,157.219
C00728=1036.044,-84.176,420.624,168.270,38.542,157.219
C00729=1036.052,-83.858,420.610,168.273,38.541,157.218
C00730=1036.059,-83.539,420.596,168.276,38.540,157.218
C00731=1036.066,-83.290,420.586,168.278,38.540,157.218
C00732=1036.072,-83.040,420.575,168.281,38.539,157.218
C00733=1036.078,-82.791,420.564,168.284,38.539,157.218
C00734=1036.085,-82.541,420.553,168.286,38.538,157.218
C00735=1036.091,-82.291,420.543,168.289,38.537,157.218
C00736=1036.097,-82.041,420.531,168.292,38.537,157.218
C00737=1036.103,-81.792,420.521,168.294,38.536,157.218
C00738=1036.109,-81.542,420.510,168.297,38.535,157.218
C00739=1036.116,-81.292,420.499,168.300,38.534,157.218
C00740=1036.122,-81.043,420.489,168.302,38.534,157.218
C00741=1036.128,-80.793,420.477,168.305,38.534,157.218
C00742=1036.134,-80.543,420.466,168.308,38.533,157.218
C00743=1036.141,-80.293,420.456,168.310,38.533,157.218
C00744=1036.147,-80.044,420.445,168.313,38.532,157.218
C00745=1036.153,-79.794,420.434,168.316,38.531,157.218
C00746=1036.159,-79.544,420.423,168.318,38.531,157.218
C00747=1036.165,-79.295,420.412,168.320,38.530,157.218
C00748=1036.172,-79.045,420.401,168.323,38.529,157.218
C00749=1036.178,-78.796,420.390,168.325,38.529,157.218
C00750=1036.184,-78.546,420.378,168.328,38.528,157.217
C00751=1036.190,-78.296,420.368,168.330,38.528,157.217
C00752=1036.196,-78.047,420.357,168.333,38.527,157.217
C00753=1036.202,-77.797,420.345,168.336,38.527,157.217
C00754=1036.208,-77.547,420.335,168.338,38.526,157.217
C00755=1036.214,-77.298,420.323,168.341,38.526,157.217
C00756=1036.220,-77.048,420.312,168.344,38.525,157.217
C00757=1036.226,-76.798,420.301,168.346,38.525,157.217
C00758=1036.232,-76.548,420.290,168.349,38.525,157.217
C00759=1036.239,-76.298,420.278,168.351,38.524,157.217
C00760=1036.245,-76.050,420.267,168.354,38.524,157.217
C00761=1036.252,-75.799,420.256,168.357,38.523,157.217
C00762=1036.257,-75.550,420.245,168.359,38.523,157.217
C00763=1036.264,-75.300,420.234,168.362,38.522,157.217
C00764=1036.270,-75.051,420.222,168.364,38.522,157.217
C00765=1036.276,-74.801,420.211,168.367,38.521,157.217
C00766=1036.282,-74.551,420.200,168.370,38.521,157.217
C00767=1036.288,-74.301,420.189,168.372,38.520,157.217
C00768=1036.294,-74.052,420.177,168.375,38.520,157.217
C00769=1036.301,-73.802,420.166,168.377,38.519,157.217
C00770=1036.306,-73.552,420.155,168.380,38.519,157.217
C00771=1036.312,-73.303,420.143,168.383,38.519,157.217
C00772=1036.318,-73.053,420.132,168.385,38.518,157.217
C00773=1036.325,-72.804,420.120,168.388,38.518,157.217
C00774=1036.330,-72.554,420.109,168.390,38.518,157.217
C00775=1036.337,-72.304,420.098,168.393,38.517,157.217
C00776=1036.342,-72.055,420.086,168.395,38.517,157.217
C00777=1036.348,-71.804,420.074,168.398,38.517,157.217
C00778=1036.354,-71.556,420.063,168.400,38.516,157.217
C00779=1036.361,-71.305,420.052,168.402,38.516,157.217
C00780=1036.367,-71.057,420.040,168.405,38.516,157.217
C00781=1036.372,-70.806,420.028,168.407,38.515,157.217
C00782=1036.379,-70.556,420.016,168.410,38.515,157.217
C00783=1036.385,-70.307,420.005,168.412,38.515,157.217
C00784=1036.391,-70.057,419.994,168.415,38.514,157.217
C00785=1036.397,-69.808,419.982,168.417,38.514,157.217
C00786=1036.403,-69.557,419.971,168.420,38.514,157.217
C00787=1036.409,-69.309,419.959,168.422,38.513,157.217
C00788=1036.415,-69.059,419.947,168.425,38.513,157.217
C00789=1036.422,-68.809,419.936,168.428,38.512,157.217
C00790=1036.427,-68.560,419.924,168.430,38.512,157.217
C00791=1036.434,-68.277,419.911,168.433,38.512,157.217
C00792=1036.441,-67.994,419.897,168.436,38.511,157.217
C00793=1036.448,-67.711,419.884,168.439,38.511,157.217
C00794=1036.455,-67.428,419.871,168.442,38.510,157.217
C00795=1036.461,-67.179,419.859,168.444,38.510,157.217
C00796=1036.468,-66.928,419.848,168.447,38.509,157.217
C00797=1036.474,-66.680,419.836,168.449,38.509,157.217
C00798=1036.479,-66.429,419.825,168.452,38.509,157.217
C00799=1036.485,-66.180,419.813,168.454,38.508,157.217
C00800=1036.492,-65.931,419.801,168.457,38.508,157.217
C00801=1036.498,-65.680,419.790,168.459,38.508,157.217
C00802=1036.504,-65.431,419.778,168.462,38.507,157.217
C00803=1036.510,-65.182,419.766,168.465,38.507,157.217
C00804=1036.517,-64.931,419.754,168.467,38.507,157.217
C00805=1036.523,-64.682,419.743,168.470,38.506,157.217
C00806=1036.529,-64.433,419.730,168.472,38.506,157.217
C00807=1036.535,-64.183,419.719,168.475,38.506,157.217
C00808=1036.542,-63.933,419.707,168.477,38.506,157.217
C00809=1036.548,-63.684,419.696,168.480,38.505,157.217
C00810=1036.553,-63.434,419.684,168.482,38.505,157.217
C00811=1036.560,-63.184,419.672,168.485,38.505,157.217
C00812=1036.567,-62.934,419.660,168.487,38.504,157.217
C00813=1036.572,-62.685,419.648,168.490,38.504,157.217
C00814=1036.578,-62.435,419.636,168.492,38.504,157.217
C00815=1036.585,-62.185,419.624,168.495,38.504,157.217
C00816=1036.591,-61.937,419.613,168.497,38.503,157.217
C00817=1036.597,-61.687,419.600,168.500,38.503,157.217
C00818=1036.603,-61.437,419.589,168.503,38.503,157.217
C00819=1036.610,-61.187,419.577,168.505,38.502,157.217
C00820=1036.616,-60.937,419.564,168.508,38.502,157.217
C00821=1036.622,-60.688,419.553,168.510,38.502,157.217
C00822=1036.628,-60.438,419.542,168.513,38.501,157.217
C00823=1036.635,-60.188,419.530,168.515,38.501,157.217
C00824=1036.641,-59.939,419.517,168.518,38.501,157.217
C00825=1036.647,-59.689,419.505,168.520,38.500,157.217
C00826=1036.653,-59.440,419.494,168.523,38.500,157.217
C00827=1036.659,-59.190,419.481,168.525,38.500,157.217
C00828=1036.666,-58.940,419.470,168.528,38.499,157.217
C00829=1036.672,-58.690,419.458,168.530,38.499,157.217
C00830=1036.678,-58.441,419.445,168.533,38.498,157.217
C00831=1036.684,-58.192,419.434,168.535,38.498,157.217
C00832=1036.691,-57.942,419.422,168.538,38.498,157.217
C00833=1036.697,-57.692,419.409,168.540,38.498,157.217
C00834=1036.703,-57.443,419.397,168.543,38.497,157.217
C00835=1036.710,-57.193,419.385,168.545,38.497,157.217
C00836=1036.717,-56.944,419.373,168.548,38.497,157.217
C00837=1036.723,-56.694,419.361,168.550,38.497,157.217
C00838=1036.728,-56.444,419.350,168.553,38.496,157.217
C00839=1036.735,-56.195,419.338,168.555,38.496,157.217
C00840=1036.741,-55.945,419.325,168.558,38.496,157.217
C00841=1036.748,-55.695,419.313,168.560,38.495,157.217
C00842=1036.754,-55.446,419.301,168.563,38.495,157.217
C00843=1036.760,-55.196,419.289,168.565,38.495,157.217
C00844=1036.767,-54.946,419.277,168.568,38.495,157.217
C00845=1036.773,-54.697,419.265,168.570,38.494,157.217
C00846=1036.779,-54.447,419.252,168.573,38.494,157.217
C00847=1036.786,-54.197,419.240,168.575,38.494,157.217
C00848=1036.792,-53.947,419.228,168.578,38.493,157.217
C00849=1036.798,-53.698,419.216,168.579,38.493,157.217
C00850=1036.805,-53.449,419.204,168.583,38.493,157.217
C00851=1036.810,-53.199,419.192,168.585,38.492,157.217
C00852=1036.817,-52.950,419.179,168.588,38.492,157.217
C00853=1036.824,-52.700,419.167,168.589,38.492,157.217
C00854=1036.830,-52.450,419.155,168.592,38.491,157.217
C00855=1036.838,-52.169,419.141,168.595,38.491,157.217
C00856=1036.845,-51.887,419.127,168.598,38.491,157.217
C00857=1036.852,-51.605,419.113,168.600,38.490,157.217
C00858=1036.859,-51.324,419.100,168.603,38.490,157.217
C00859=1036.866,-51.075,419.087,168.606,38.490,157.217
C00860=1036.872,-50.825,419.075,168.608,38.490,157.217
C00861=1036.878,-50.576,419.063,168.611,38.489,157.217
C00862=1036.885,-50.326,419.051,168.613,38.489,157.217
C00863=1036.891,-50.076,419.038,168.615,38.489,157.217
C00864=1036.897,-49.826,419.026,168.618,38.489,157.217
C00865=1036.903,-49.577,419.012,168.620,38.489,157.217
C00866=1036.909,-49.327,419.000,168.623,38.488,157.217
C00867=1036.915,-49.077,418.988,168.625,38.488,157.217
C00868=1036.921,-48.828,418.975,168.627,38.488,157.217
C00869=1036.928,-48.579,418.963,168.631,38.488,157.217
C00870=1036.934,-48.329,418.950,168.633,38.488,157.217
C00871=1036.940,-48.079,418.938,168.636,38.488,157.217
C00872=1036.946,-47.830,418.924,168.638,38.488,157.217
C00873=1036.953,-47.580,418.912,168.641,38.488,157.217
C00874=1036.959,-47.330,418.900,168.643,38.487,157.217
C00875=1036.965,-47.081,418.887,168.645,38.487,157.217
C00876=1036.972,-46.831,418.875,168.648,38.487,157.217
C00877=1036.978,-46.581,418.862,168.650,38.487,157.217
C00878=1036.984,-46.332,418.849,168.653,38.487,157.218
C00879=1036.990,-46.082,418.836,168.655,38.487,157.218
C00880=1036.996,-45.833,418.824,168.657,38.487,157.218
C00881=1037.003,-45.583,418.811,168.660,38.487,157.218
C00882=1037.008,-45.334,418.798,168.662,38.487,157.218
C00883=1037.014,-45.084,418.786,168.665,38.486,157.218
C00884=1037.021,-44.835,418.773,168.667,38.486,157.218
C00885=1037.027,-44.585,418.761,168.669,38.486,157.218
C00886=1037.033,-44.336,418.747,168.672,38.486,157.218
C00887=1037.040,-44.085,418.734,168.674,38.486,157.218
C00888=1037.047,-43.836,418.722,168.677,38.486,157.218
C00889=1037.053,-43.586,418.709,168.679,38.486,157.218
C00890=1037.059,-43.336,418.697,168.681,38.486,157.218
C00891=1037.065,-43.087,418.683,168.684,38.485,157.218
C00892=1037.072,-42.837,418.671,168.686,38.485,157.218
C00893=1037.078,-42.588,418.658,168.689,38.485,157.218
C00894=1037.084,-42.338,418.646,168.691,38.486,157.218
C00895=1037.090,-42.089,418.632,168.693,38.486,157.218
C00896=1037.097,-41.839,418.620,168.696,38.485,157.218
C00897=1037.103,-41.590,418.607,168.698,38.485,157.218
C00898=1037.109,-41.340,418.594,168.701,38.485,157.218
C00899=1037.115,-41.090,418.581,168.703,38.485,157.218
C00900=1037.121,-40.840,418.568,168.705,38.485,157.218
C00901=1037.128,-40.592,418.556,168.708,38.485,157.218
C00902=1037.134,-40.342,418.543,168.710,38.485,157.218
C00903=1037.141,-40.092,418.530,168.713,38.485,157.218
C00904=1037.147,-39.842,418.516,168.715,38.484,157.218
C00905=1037.154,-39.593,418.504,168.717,38.484,157.218
C00906=1037.160,-39.344,418.491,168.720,38.484,157.219
C00907=1037.166,-39.094,418.478,168.722,38.484,157.219
C00908=1037.172,-38.844,418.465,168.725,38.484,157.219
C00909=1037.179,-38.594,418.452,168.727,38.484,157.219
C00910=1037.185,-38.345,418.439,168.729,38.484,157.219
C00911=1037.191,-38.095,418.426,168.732,38.484,157.219
C00912=1037.197,-37.846,418.412,168.734,38.483,157.219
C00913=1037.203,-37.596,418.400,168.736,38.484,157.219
C00914=1037.210,-37.347,418.387,168.739,38.484,157.219
C00915=1037.216,-37.097,418.373,168.741,38.484,157.219
C00916=1037.222,-36.847,418.360,168.743,38.484,157.219
C00917=1037.228,-36.598,418.347,168.747,38.483,157.219
C00918=1037.235,-36.349,418.334,168.749,38.484,157.219
C00919=1037.242,-36.067,418.319,168.752,38.484,157.219
C00920=1037.249,-35.786,418.304,168.754,38.484,157.219
C00921=1037.256,-35.505,418.290,168.757,38.484,157.219
C00922=1037.262,-35.224,418.275,168.759,38.484,157.219
C00923=1037.269,-34.974,418.261,168.762,38.484,157.219
C00924=1037.275,-34.724,418.248,168.764,38.484,157.219
C00925=1037.282,-34.475,418.234,168.766,38.484,157.219
C00926=1037.288,-34.226,418.221,168.769,38.484,157.219
C00927=1037.294,-33.976,418.209,168.771,38.484,157.220
C00928=1037.300,-33.727,418.195,168.773,38.483,157.220
C00929=1037.307,-33.477,418.182,168.776,38.484,157.220
C00930=1037.313,-33.227,418.168,168.778,38.484,157.220
C00931=1037.319,-32.978,418.155,168.780,38.484,157.220
C00932=1037.326,-32.728,418.142,168.783,38.484,157.220
C00933=1037.332,-32.478,418.129,168.785,38.483,157.220
C00934=1037.338,-32.229,418.116,168.787,38.484,157.220
C00935=1037.344,-31.980,418.102,168.790,38.484,157.220
C00936=1037.351,-31.730,418.089,168.792,38.484,157.220
C00937=1037.357,-31.481,418.076,168.794,38.484,157.220
C00938=1037.364,-31.231,418.062,168.797,38.484,157.220
C00939=1037.370,-30.981,418.049,168.799,38.483,157.220
C00940=1037.377,-30.732,418.035,168.801,38.484,157.220
C00941=1037.382,-30.482,418.022,168.804,38.484,157.220
C00942=1037.389,-30.232,418.009,168.806,38.484,157.220
C00943=1037.395,-29.983,417.995,168.808,38.484,157.220
C00944=1037.401,-29.733,417.982,168.810,38.484,157.220
C00945=1037.408,-29.483,417.968,168.814,38.484,157.221
C00946=1037.414,-29.234,417.955,168.816,38.484,157.221
C00947=1037.420,-28.985,417.942,168.818,38.484,157.221
C00948=1037.427,-28.735,417.928,168.821,38.484,157.221
C00949=1037.433,-28.486,417.915,168.823,38.484,157.221
C00950=1037.439,-28.236,417.902,168.825,38.483,157.221
C00951=1037.446,-27.986,417.888,168.828,38.484,157.221
C00952=1037.453,-27.737,417.875,168.830,38.484,157.221
C00953=1037.458,-27.488,417.861,168.832,38.484,157.221
C00954=1037.465,-27.238,417.847,168.835,38.484,157.221
C00955=1037.471,-26.988,417.834,168.837,38.483,157.221
C00956=1037.478,-26.738,417.820,168.839,38.484,157.221
C00957=1037.483,-26.489,417.807,168.841,38.484,157.221
C00958=1037.490,-26.240,417.793,168.844,38.484,157.221
C00959=1037.496,-25.990,417.780,168.846,38.484,157.221
C00960=1037.502,-25.741,417.765,168.848,38.484,157.221
C00961=1037.509,-25.491,417.751,168.850,38.484,157.221
C00962=1037.515,-25.241,417.738,168.853,38.485,157.222
C00963=1037.521,-24.992,417.724,168.855,38.484,157.222
C00964=1037.527,-24.742,417.711,168.857,38.484,157.222
C00965=1037.534,-24.493,417.697,168.859,38.485,157.222
C00966=1037.539,-24.243,417.684,168.862,38.485,157.222
C00967=1037.546,-23.994,417.669,168.865,38.485,157.222
C00968=1037.552,-23.744,417.656,168.867,38.485,157.222
C00969=1037.559,-23.494,417.642,168.869,38.485,157.222
C00970=1037.565,-23.245,417.628,168.872,38.486,157.222
C00971=1037.572,-22.995,417.615,168.874,38.486,157.222
C00972=1037.577,-22.746,417.600,168.876,38.485,157.222
C00973=1037.584,-22.497,417.587,168.878,38.486,157.222
C00974=1037.590,-22.247,417.573,168.881,38.486,157.222
C00975=1037.596,-21.997,417.559,168.883,38.486,157.222
C00976=1037.603,-21.748,417.545,168.885,38.486,157.223
C00977=1037.609,-21.499,417.532,168.887,38.486,157.223
C00978=1037.615,-21.248,417.518,168.890,38.486,157.223
C00979=1037.621,-20.999,417.504,168.892,38.487,157.223
C00980=1037.629,-20.750,417.490,168.894,38.486,157.223
C00981=1037.634,-20.500,417.476,168.896,38.486,157.223
C00982=1037.641,-20.250,417.462,168.898,38.487,157.223
C00983=1037.648,-19.969,417.447,168.901,38.487,157.223
C00984=1037.655,-19.687,417.431,168.904,38.487,157.223
C00985=1037.663,-19.405,417.415,168.907,38.487,157.223
C00986=1037.669,-19.124,417.399,168.910,38.487,157.223
C00987=1037.676,-18.873,417.385,168.912,38.487,157.223
C00988=1037.682,-18.624,417.372,168.914,38.487,157.223
C00989=1037.688,-18.374,417.357,168.916,38.487,157.223
C00990=1037.694,-18.125,417.344,168.919,38.487,157.223
C00991=1037.701,-17.875,417.330,168.921,38.488,157.224
C00992=1037.707,-17.626,417.316,168.923,38.488,157.224
C00993=1037.714,-17.376,417.302,168.925,38.487,157.224
C00994=1037.720,-17.128,417.288,168.927,38.488,157.224
C00995=1037.726,-16.877,417.274,168.930,38.488,157.224
C00996=1037.733,-16.627,417.260,168.932,38.488,157.224
C00997=1037.739,-16.378,417.245,168.934,38.488,157.224
C00998=1037.746,-16.128,417.232,168.936,38.488,157.224
C00999=1037.752,-15.880,417.218,168.939,38.488,157.224
C01000=1037.758,-15.630,417.204,168.941,38.489,157.224
C01001=1037.765,-15.380,417.190,168.943,38.488,157.224
C01002=1037.771,-15.131,417.175,168.945,38.489,157.224
C01003=1037.777,-14.880,417.161,168.947,38.489,157.224
C01004=1037.784,-14.632,417.147,168.951,38.489,157.225
C01005=1037.790,-14.382,417.132,168.953,38.489,157.225
C01006=1037.796,-14.133,417.119,168.955,38.490,157.225
C01007=1037.803,-13.883,417.104,168.957,38.490,157.225
C01008=1037.808,-13.634,417.090,168.959,38.490,157.225
C01009=1037.815,-13.384,417.076,168.961,38.490,157.225
C01010=1037.821,-13.134,417.062,168.964,38.490,157.225
C01011=1037.827,-12.885,417.047,168.966,38.491,157.225
C01012=1037.834,-12.635,417.033,168.968,38.491,157.225
C01013=1037.840,-12.386,417.019,168.970,38.491,157.225
C01014=1037.846,-12.136,417.004,168.972,38.491,157.225
C01015=1037.853,-11.886,416.990,168.974,38.491,157.225
C01016=1037.859,-11.637,416.976,168.977,38.491,157.226
C01017=1037.865,-11.388,416.961,168.979,38.492,157.226
C01018=1037.871,-11.139,416.947,168.981,38.492,157.226
C01019=1037.878,-10.889,416.932,168.984,38.492,157.226
C01020=1037.884,-10.639,416.919,168.986,38.492,157.226
C01021=1037.890,-10.390,416.904,168.988,38.493,157.226
C01022=1037.897,-10.140,416.889,168.991,38.493,157.226
C01023=1037.903,-9.890,416.876,168.993,38.493,157.226
C01024=1037.909,-9.641,416.861,168.995,38.493,157.226
C01025=1037.916,-9.392,416.846,168.997,38.494,157.226
C01026=1037.923,-9.142,416.832,168.999,38.493,157.226
C01027=1037.928,-8.893,416.818,169.001,38.494,157.227
C01028=1037.935,-8.643,416.803,169.004,38.494,157.227
C01029=1037.942,-8.394,416.789,169.006,38.494,157.227
C01030=1037.947,-8.144,416.775,169.008,38.494,157.227
C01031=1037.954,-7.895,416.760,169.010,38.494,157.227
C01032=1037.960,-7.645,416.745,169.012,38.495,157.227
C01033=1037.966,-7.396,416.731,169.014,38.495,157.227
C01034=1037.972,-7.146,416.717,169.017,38.495,157.227
C01035=1037.979,-6.896,416.702,169.019,38.495,157.227
C01036=1037.985,-6.648,416.688,169.022,38.496,157.227
C01037=1037.992,-6.398,416.673,169.024,38.495,157.227
C01038=1037.998,-6.148,416.658,169.026,38.496,157.227
C01039=1038.005,-5.898,416.644,169.028,38.496,157.227
C01040=1038.011,-5.649,416.630,169.030,38.496,157.228
C01041=1038.017,-5.400,416.615,169.033,38.496,157.228
C01042=1038.024,-5.150,416.600,169.035,38.497,157.228
C01043=1038.031,-4.901,416.585,169.037,38.497,157.228
C01044=1038.036,-4.651,416.572,169.039,38.497,157.228
C01045=1038.043,-4.402,416.557,169.041,38.497,157.228
C01046=1038.050,-4.152,416.542,169.043,38.497,157.228
C01047=1038.057,-3.869,416.526,169.046,38.498,157.228
C01048=1038.064,-3.586,416.509,169.048,38.497,157.228
C01049=1038.070,-3.302,416.492,169.051,38.498,157.228
C01050=1038.078,-3.018,416.475,169.054,38.499,157.229
C01051=1038.084,-2.769,416.461,169.056,38.499,157.229
C01052=1038.090,-2.519,416.446,169.058,38.499,157.229
C01053=1038.097,-2.270,416.431,169.060,38.499,157.229
C01054=1038.103,-2.020,416.416,169.062,38.500,157.229
C01055=1038.109,-1.771,416.401,169.064,38.500,157.229
C01056=1038.115,-1.521,416.386,169.066,38.500,157.229
C01057=1038.122,-1.272,416.371,169.069,38.501,157.229
C01058=1038.128,-1.022,416.356,169.071,38.501,157.229
C01059=1038.134,-0.773,416.342,169.073,38.501,157.229
C01060=1038.140,-0.523,416.327,169.075,38.501,157.230
C01061=1038.147,-0.274,416.312,169.077,38.502,157.230
C01062=1038.153,-0.024,416.297,169.080,38.502,157.230
C01063=1038.159,0.225,416.282,169.082,38.502,157.230
C01064=1038.165,0.474,416.267,169.084,38.503,157.230
C01065=1038.171,0.724,416.252,169.086,38.503,157.230
C01066=1038.178,0.973,416.237,169.088,38.503,157.230
C01067=1038.185,1.223,416.222,169.090,38.504,157.230
C01068=1038.190,1.472,416.207,169.092,38.504,157.230
C01069=1038.197,1.721,416.192,169.095,38.504,157.230
C01070=1038.203,1.971,416.177,169.097,38.505,157.231
C01071=1038.209,2.221,416.162,169.099,38.505,157.231
C01072=1038.216,2.470,416.147,169.101,38.505,157.231
C01073=1038.222,2.720,416.133,169.104,38.506,157.231
C01074=1038.227,2.969,416.117,169.106,38.506,157.231
C01075=1038.234,3.218,416.102,169.108,38.506,157.231
C01076=1038.240,3.468,416.087,169.110,38.507,157.231
C01077=1038.247,3.718,416.072,169.112,38.507,157.231
C01078=1038.253,3.967,416.057,169.114,38.507,157.231
C01079=1038.259,4.217,416.042,169.116,38.508,157.232
C01080=1038.266,4.467,416.027,169.118,38.508,157.232
C01081=1038.272,4.715,416.012,169.120,38.508,157.232
C01082=1038.278,4.965,415.997,169.123,38.509,157.232
C01083=1038.285,5.214,415.982,169.125,38.508,157.232
C01084=1038.291,5.464,415.967,169.127,38.509,157.232
C01085=1038.298,5.713,415.951,169.129,38.509,157.232
C01086=1038.304,5.963,415.936,169.132,38.509,157.232
C01087=1038.311,6.212,415.921,169.134,38.510,157.232
C01088=1038.317,6.462,415.906,169.136,38.510,157.232
C01089=1038.324,6.711,415.891,169.138,38.510,157.233
C01090=1038.329,6.960,415.875,169.140,38.511,157.233
C01091=1038.335,7.210,415.861,169.142,38.511,157.233
C01092=1038.341,7.460,415.846,169.144,38.511,157.233
C01093=1038.348,7.709,415.830,169.146,38.511,157.233
C01094=1038.355,7.958,415.815,169.148,38.512,157.233
C01095=1038.361,8.208,415.800,169.150,38.512,157.233
C01096=1038.368,8.457,415.784,169.152,38.512,157.233
C01097=1038.374,8.707,415.769,169.154,38.513,157.233
C01098=1038.380,8.956,415.754,169.157,38.513,157.233
C01099=1038.387,9.206,415.740,169.160,38.513,157.234
C01100=1038.393,9.455,415.724,169.162,38.514,157.234
C01101=1038.399,9.705,415.708,169.164,38.514,157.234
C01102=1038.406,9.954,415.693,169.166,38.514,157.234
C01103=1038.412,10.204,415.678,169.168,38.514,157.234
C01104=1038.419,10.453,415.663,169.170,38.515,157.234
C01105=1038.425,10.702,415.647,169.172,38.515,157.234
C01106=1038.432,10.952,415.632,169.174,38.515,157.234
C01107=1038.438,11.202,415.617,169.176,38.516,157.234
C01108=1038.445,11.451,415.602,169.178,38.516,157.234
C01109=1038.451,11.700,415.587,169.180,38.516,157.235
C01110=1038.458,11.949,415.571,169.183,38.517,157.235
C01111=1038.464,12.236,415.553,169.186,38.516,157.235
C01112=1038.472,12.521,415.536,169.188,38.517,157.235
C01113=1038.479,12.806,415.518,169.190,38.518,157.235
C01114=1038.487,13.091,415.500,169.193,38.517,157.235
C01115=1038.493,13.341,415.485,169.195,38.518,157.235
C01116=1038.500,13.590,415.470,169.197,38.518,157.235
C01117=1038.506,13.840,415.455,169.199,38.518,157.235
C01118=1038.513,14.089,415.439,169.201,38.519,157.236
C01119=1038.519,14.339,415.424,169.203,38.519,157.236
C01120=1038.525,14.588,415.408,169.205,38.519,157.236
C01121=1038.532,14.837,415.393,169.207,38.520,157.236
C01122=1038.538,15.087,415.377,169.210,38.520,157.236
C01123=1038.544,15.336,415.362,169.212,38.521,157.236
C01124=1038.551,15.585,415.346,169.214,38.521,157.236
C01125=1038.556,15.835,415.331,169.216,38.521,157.236
C01126=1038.563,16.084,415.315,169.218,38.522,157.236
C01127=1038.569,16.334,415.299,169.220,38.522,157.237
C01128=1038.575,16.583,415.284,169.222,38.522,157.237
C01129=1038.582,16.832,415.268,169.224,38.523,157.237
C01130=1038.588,17.082,415.252,169.226,38.523,157.237
C01131=1038.594,17.331,415.237,169.228,38.523,157.237
C01132=1038.602,17.581,415.221,169.230,38.524,157.237
C01133=1038.607,17.831,415.205,169.233,38.524,157.237
C01134=1038.614,18.080,415.190,169.235,38.525,157.237
C01135=1038.620,18.329,415.173,169.237,38.525,157.237
C01136=1038.626,18.579,415.158,169.239,38.525,157.238
C01137=1038.633,18.828,415.143,169.241,38.526,157.238
C01138=1038.639,19.077,415.126,169.243,38.526,157.238
C01139=1038.645,19.327,415.112,169.245,38.526,157.238
C01140=1038.651,19.576,415.095,169.247,38.527,157.238
C01141=1038.658,19.825,415.080,169.249,38.527,157.238
C01142=1038.665,20.075,415.064,169.251,38.527,157.238
C01143=1038.671,20.325,415.048,169.253,38.528,157.238
C01144=1038.678,20.574,415.032,169.256,38.528,157.239
C01145=1038.684,20.824,415.016,169.258,38.529,157.239
C01146=1038.690,21.073,415.000,169.260,38.529,157.239
C01147=1038.696,21.323,414.985,169.262,38.529,157.239
C01148=1038.702,21.572,414.969,169.264,38.530,157.239
C01149=1038.709,21.821,414.953,169.266,38.530,157.239
C01150=1038.715,22.070,414.937,169.268,38.531,157.239
C01151=1038.722,22.320,414.921,169.270,38.531,157.239
C01152=1038.727,22.570,414.905,169.272,38.531,157.239
C01153=1038.734,22.819,414.890,169.274,38.532,157.240
C01154=1038.740,23.068,414.873,169.277,38.532,157.240
C01155=1038.747,23.317,414.858,169.279,38.533,157.240
C01156=1038.753,23.567,414.841,169.281,38.533,157.240
C01157=1038.759,23.816,414.826,169.283,38.533,157.240
C01158=1038.766,24.067,414.810,169.285,38.534,157.240
C01159=1038.772,24.316,414.794,169.287,38.535,157.240
C01160=1038.778,24.565,414.778,169.289,38.534,157.240
C01161=1038.785,24.814,414.762,169.290,38.535,157.241
C01162=1038.791,25.063,414.746,169.292,38.536,157.241
C01163=1038.798,25.313,414.729,169.294,38.536,157.241
C01164=1038.804,25.562,414.714,169.297,38.536,157.241
C01165=1038.810,25.812,414.697,169.299,38.536,157.241
C01166=1038.817,26.061,414.682,169.301,38.537,157.241
C01167=1038.823,26.310,414.665,169.303,38.538,157.241
C01168=1038.830,26.560,414.650,169.305,38.538,157.241
C01169=1038.836,26.810,414.634,169.307,38.538,157.241
C01170=1038.842,27.059,414.618,169.309,38.539,157.242
C01171=1038.848,27.308,414.602,169.311,38.539,157.242
C01172=1038.854,27.558,414.586,169.313,38.540,157.242
C01173=1038.862,27.807,414.570,169.315,38.540,157.242
C01174=1038.868,28.057,414.553,169.318,38.540,157.242
C01175=1038.875,28.343,414.535,169.320,38.541,157.242
C01176=1038.882,28.629,414.516,169.323,38.541,157.242
C01177=1038.889,28.917,414.497,169.325,38.542,157.243
C01178=1038.897,29.203,414.479,169.327,38.542,157.243
C01179=1038.903,29.453,414.462,169.329,38.543,157.243
C01180=1038.909,29.702,414.446,169.331,38.543,157.243
C01181=1038.915,29.951,414.430,169.333,38.544,157.243
C01182=1038.922,30.201,414.414,169.336,38.544,157.243
C01183=1038.928,30.450,414.398,169.338,38.544,157.243
C01184=1038.934,30.700,414.381,169.340,38.545,157.243
C01185=1038.941,30.948,414.365,169.342,38.545,157.244
C01186=1038.947,31.198,414.348,169.343,38.546,157.244
C01187=1038.953,31.448,414.332,169.345,38.546,157.244
C01188=1038.959,31.697,414.316,169.347,38.547,157.244
C01189=1038.965,31.946,414.300,169.349,38.547,157.244
C01190=1038.972,32.196,414.284,169.351,38.547,157.244
C01191=1038.978,32.445,414.267,169.353,38.548,157.244
C01192=1038.985,32.694,414.250,169.356,38.548,157.245
C01193=1038.991,32.944,414.234,169.358,38.549,157.245
C01194=1038.997,33.193,414.217,169.360,38.549,157.245
C01195=1039.004,33.442,414.202,169.362,38.550,157.245
C01196=1039.010,33.693,414.185,169.364,38.551,157.245
C01197=1039.016,33.942,414.169,169.366,38.550,157.245
C01198=1039.023,34.191,414.152,169.368,38.551,157.245
C01199=1039.029,34.440,414.136,169.370,38.552,157.245
C01200=1039.036,34.690,414.120,169.372,38.552,157.246
C01201=1039.042,34.939,414.103,169.375,38.553,157.246
C01202=1039.048,35.188,414.086,169.376,38.553,157.246
C01203=1039.055,35.438,414.070,169.378,38.553,157.246
C01204=1039.061,35.687,414.054,169.380,38.554,157.246
C01205=1039.067,35.936,414.038,169.382,38.554,157.246
C01206=1039.074,36.186,414.021,169.384,38.555,157.246
C01207=1039.080,36.435,414.004,169.386,38.555,157.246
C01208=1039.087,36.685,413.988,169.388,38.556,157.247
C01209=1039.093,36.934,413.971,169.390,38.556,157.247
C01210=1039.100,37.183,413.955,169.392,38.556,157.247
C01211=1039.106,37.433,413.938,169.395,38.557,157.247
C01212=1039.112,37.682,413.922,169.397,38.557,157.247
C01213=1039.118,37.931,413.905,169.399,38.558,157.247
C01214=1039.125,38.181,413.889,169.401,38.558,157.247
C01215=1039.131,38.430,413.872,169.402,38.559,157.248
C01216=1039.137,38.679,413.855,169.404,38.559,157.248
C01217=1039.144,38.929,413.839,169.406,38.560,157.248
C01218=1039.149,39.178,413.821,169.408,38.560,157.248
C01219=1039.156,39.428,413.805,169.411,38.561,157.248
C01220=1039.162,39.678,413.788,169.413,38.561,157.248
C01221=1039.168,39.926,413.771,169.415,38.561,157.248
C01222=1039.174,40.176,413.755,169.417,38.562,157.248
C01223=1039.181,40.425,413.738,169.419,38.563,157.249
C01224=1039.187,40.674,413.721,169.421,38.563,157.249
C01225=1039.194,40.924,413.704,169.422,38.564,157.249
C01226=1039.199,41.173,413.688,169.424,38.564,157.249
C01227=1039.206,41.423,413.670,169.426,38.565,157.249
C01228=1039.212,41.672,413.654,169.429,38.565,157.249
C01229=1039.219,41.921,413.637,169.431,38.566,157.249
C01230=1039.225,42.171,413.621,169.433,38.566,157.250
C01231=1039.231,42.419,413.604,169.435,38.567,157.250
C01232=1039.238,42.670,413.587,169.437,38.567,157.250
C01233=1039.244,42.918,413.570,169.439,38.567,157.250
C01234=1039.251,43.168,413.553,169.441,38.568,157.250
C01235=1039.257,43.417,413.536,169.442,38.568,157.250
C01236=1039.262,43.667,413.520,169.444,38.569,157.250
C01237=1039.269,43.916,413.502,169.446,38.569,157.251
C01238=1039.275,44.165,413.486,169.449,38.571,157.251
C01239=1039.283,44.452,413.466,169.451,38.571,157.251
C01240=1039.289,44.739,413.446,169.453,38.572,157.251
C01241=1039.296,45.025,413.427,169.455,38.572,157.251
C01242=1039.303,45.312,413.407,169.458,38.573,157.251
C01243=1039.309,45.561,413.391,169.459,38.573,157.252
C01244=1039.316,45.811,413.373,169.461,38.574,157.252
C01245=1039.322,46.060,413.356,169.464,38.574,157.252
C01246=1039.328,46.309,413.340,169.466,38.576,157.252
C01247=1039.335,46.558,413.322,169.468,38.576,157.252
C01248=1039.340,46.808,413.305,169.470,38.577,157.252
C01249=1039.347,47.058,413.288,169.472,38.577,157.253
C01250=1039.353,47.306,413.271,169.474,38.578,157.253
C01251=1039.359,47.556,413.253,169.475,38.578,157.253
C01252=1039.365,47.805,413.236,169.478,38.579,157.253
C01253=1039.372,48.055,413.219,169.480,38.579,157.253
C01254=1039.377,48.304,413.202,169.482,38.580,157.253
C01255=1039.384,48.553,413.185,169.484,38.580,157.253
C01256=1039.390,48.803,413.168,169.486,38.581,157.254
C01257=1039.396,49.052,413.150,169.488,38.581,157.254
C01258=1039.403,49.301,413.133,169.489,38.582,157.254
C01259=1039.409,49.551,413.116,169.491,38.583,157.254
C01260=1039.415,49.800,413.099,169.494,38.583,157.254
C01261=1039.421,50.050,413.082,169.496,38.584,157.254
C01262=1039.428,50.298,413.065,169.498,38.584,157.254
C01263=1039.435,50.548,413.048,169.500,38.585,157.255
C01264=1039.440,50.797,413.030,169.502,38.585,157.255
C01265=1039.447,51.047,413.013,169.503,38.586,157.255
C01266=1039.452,51.296,412.996,169.505,38.586,157.255
C01267=1039.459,51.545,412.978,169.507,38.587,157.255
C01268=1039.465,51.794,412.962,169.510,38.587,157.255
C01269=1039.471,52.044,412.944,169.512,38.588,157.255
C01270=1039.478,52.293,412.927,169.514,38.588,157.256
C01271=1039.484,52.543,412.910,169.516,38.589,157.256
C01272=1039.490,52.792,412.892,169.518,38.590,157.256
C01273=1039.497,53.041,412.875,169.519,38.590,157.256
C01274=1039.503,53.291,412.858,169.521,38.591,157.256
C01275=1039.509,53.540,412.840,169.523,38.591,157.256
C01276=1039.516,53.789,412.823,169.526,38.592,157.257
C01277=1039.522,54.038,412.806,169.528,38.592,157.257
C01278=1039.528,54.287,412.788,169.530,38.593,157.257
C01279=1039.535,54.537,412.771,169.532,38.593,157.257
C01280=1039.541,54.786,412.754,169.534,38.594,157.257
C01281=1039.547,55.036,412.736,169.535,38.594,157.257
C01282=1039.553,55.285,412.719,169.537,38.595,157.257
C01283=1039.560,55.534,412.702,169.539,38.595,157.258
C01284=1039.566,55.784,412.684,169.542,38.596,157.258
C01285=1039.573,56.033,412.667,169.544,38.597,157.258
C01286=1039.579,56.282,412.649,169.546,38.596,157.258
C01287=1039.585,56.531,412.632,169.548,38.597,157.258
C01288=1039.592,56.780,412.615,169.550,38.597,157.258
C01289=1039.598,57.030,412.597,169.551,38.598,157.258
C01290=1039.604,57.279,412.580,169.553,38.599,157.258
C01291=1039.611,57.528,412.563,169.555,38.599,157.259
C01292=1039.617,57.778,412.545,169.557,38.600,157.259
C01293=1039.623,58.027,412.528,169.560,38.600,157.259
C01294=1039.630,58.277,412.510,169.562,38.601,157.259
C01295=1039.636,58.526,412.493,169.564,38.601,157.259
C01296=1039.643,58.775,412.476,169.566,38.602,157.259
C01297=1039.649,59.025,412.458,169.567,38.602,157.259
C01298=1039.656,59.274,412.440,169.569,38.603,157.260
C01299=1039.661,59.523,412.423,169.571,38.603,157.260
C01300=1039.668,59.772,412.405,169.573,38.604,157.260
C01301=1039.675,60.022,412.388,169.576,38.604,157.260
C01302=1039.681,60.272,412.370,169.578,38.605,157.260
C01303=1039.688,60.558,412.350,169.580,38.606,157.260
C01304=1039.696,60.844,412.330,169.582,38.606,157.261
C01305=1039.703,61.130,412.310,169.584,38.607,157.261
C01306=1039.711,61.416,412.290,169.586,38.607,157.261
C01307=1039.717,61.665,412.272,169.588,38.608,157.261
C01308=1039.724,61.914,412.255,169.590,38.608,157.261
C01309=1039.730,62.164,412.237,169.593,38.609,157.261
C01310=1039.737,62.413,412.219,169.595,38.609,157.261
C01311=1039.743,62.662,412.202,169.597,38.609,157.261
C01312=1039.749,62.912,412.184,169.599,38.610,157.262
C01313=1039.756,63.161,412.167,169.601,38.610,157.262
C01314=1039.762,63.411,412.149,169.603,38.611,157.262
C01315=1039.768,63.659,412.131,169.604,38.611,157.262
C01316=1039.775,63.909,412.113,169.606,38.612,157.262
C01317=1039.781,64.158,412.096,169.608,38.612,157.262
C01318=1039.788,64.408,412.078,169.611,38.613,157.262
C01319=1039.793,64.657,412.060,169.613,38.613,157.263
C01320=1039.800,64.906,412.043,169.615,38.614,157.263
C01321=1039.806,65.156,412.025,169.617,38.614,157.263
C01322=1039.812,65.405,412.007,169.618,38.615,157.263
C01323=1039.819,65.654,411.989,169.620,38.616,157.263
C01324=1039.825,65.903,411.971,169.622,38.616,157.263
C01325=1039.831,66.153,411.953,169.625,38.617,157.264
C01326=1039.838,66.402,411.935,169.627,38.618,157.264
C01327=1039.844,66.651,411.918,169.629,38.618,157.264
C01328=1039.850,66.901,411.900,169.630,38.619,157.264
C01329=1039.857,67.150,411.882,169.632,38.619,157.264
C01330=1039.863,67.399,411.864,169.634,38.620,157.264
C01331=1039.869,67.648,411.846,169.636,38.620,157.265
C01332=1039.875,67.897,411.827,169.638,38.621,157.265
C01333=1039.882,68.147,411.810,169.641,38.621,157.265
C01334=1039.888,68.397,411.792,169.643,38.622,157.265
C01335=1039.895,68.646,411.773,169.644,38.623,157.265
C01336=1039.900,68.895,411.756,169.646,38.623,157.265
C01337=1039.907,69.144,411.739,169.648,38.624,157.265
C01338=1039.913,69.393,411.720,169.650,38.624,157.266
C01339=1039.920,69.643,411.702,169.652,38.625,157.266
C01340=1039.926,69.892,411.683,169.655,38.626,157.266
C01341=1039.932,70.141,411.666,169.656,38.626,157.266
C01342=1039.938,70.390,411.647,169.658,38.627,157.266
C01343=1039.945,70.640,411.630,169.660,38.628,157.266
C01344=1039.951,70.889,411.611,169.662,38.628,157.267
C01345=1039.957,71.139,411.593,169.664,38.629,157.267
C01346=1039.963,71.387,411.575,169.666,38.629,157.267
C01347=1039.969,71.637,411.557,169.667,38.630,157.267
C01348=1039.976,71.886,411.538,169.669,38.630,157.267
C01349=1039.982,72.136,411.520,169.672,38.631,157.267
C01350=1039.988,72.385,411.502,169.674,38.632,157.268
C01351=1039.995,72.633,411.485,169.676,38.632,157.268
C01352=1040.001,72.883,411.466,169.678,38.633,157.268
C01353=1040.007,73.132,411.448,169.679,38.634,157.268
C01354=1040.014,73.381,411.430,169.681,38.634,157.268
C01355=1040.020,73.631,411.412,169.683,38.635,157.268
C01356=1040.026,73.880,411.393,169.686,38.635,157.268
C01357=1040.032,74.129,411.375,169.688,38.636,157.269
C01358=1040.038,74.378,411.357,169.690,38.636,157.269
C01359=1040.044,74.628,411.338,169.692,38.637,157.269
C01360=1040.051,74.877,411.320,169.693,38.638,157.269
C01361=1040.057,75.126,411.302,169.695,38.638,157.269
C01362=1040.063,75.376,411.283,169.697,38.639,157.269
C01363=1040.070,75.625,411.266,169.700,38.639,157.270
C01364=1040.077,75.874,411.247,169.702,38.640,157.270
C01365=1040.082,76.123,411.229,169.704,38.640,157.270
C01366=1040.089,76.372,411.211,169.705,38.641,157.270
C01367=1040.096,76.659,411.189,169.708,38.642,157.270
C01368=1040.104,76.945,411.168,169.710,38.643,157.271
C01369=1040.110,77.231,411.147,169.712,38.643,157.271
C01370=1040.118,77.517,411.126,169.715,38.644,157.271
C01371=1040.124,77.766,411.108,169.717,38.644,157.271
C01372=1040.131,78.015,411.089,169.719,38.645,157.271
C01373=1040.137,78.265,411.071,169.720,38.646,157.271
C01374=1040.142,78.514,411.052,169.722,38.647,157.272
C01375=1040.148,78.763,411.034,169.724,38.647,157.272
C01376=1040.155,79.012,411.015,169.726,38.648,157.272
C01377=1040.161,79.262,410.997,169.729,38.648,157.272
C01378=1040.167,79.511,410.978,169.731,38.649,157.272
C01379=1040.174,79.760,410.960,169.732,38.650,157.272
C01380=1040.179,80.009,410.941,169.734,38.650,157.273
C01381=1040.186,80.258,410.922,169.736,38.651,157.273
C01382=1040.192,80.508,410.904,169.738,38.651,157.273
C01383=1040.198,80.757,410.885,169.741,38.653,157.273
C01384=1040.205,81.006,410.867,169.742,38.653,157.273
C01385=1040.210,81.256,410.847,169.744,38.654,157.273
C01386=1040.216,81.504,410.829,169.746,38.654,157.274
C01387=1040.223,81.753,410.811,169.748,38.655,157.274
C01388=1040.229,82.003,410.793,169.750,38.656,157.274
C01389=1040.235,82.252,410.774,169.752,38.656,157.274
C01390=1040.242,82.501,410.755,169.754,38.657,157.274
C01391=1040.247,82.751,410.736,169.756,38.658,157.274
C01392=1040.254,83.000,410.717,169.758,38.658,157.275
C01393=1040.260,83.249,410.699,169.760,38.659,157.275
C01394=1040.267,83.498,410.680,169.762,38.660,157.275
C01395=1040.273,83.747,410.661,169.764,38.660,157.275
C01396=1040.279,83.997,410.642,169.765,38.661,157.275
C01397=1040.285,84.246,410.624,169.768,38.661,157.275
C01398=1040.292,84.495,410.605,169.770,38.662,157.276
C01399=1040.298,84.745,410.587,169.772,38.663,157.276
C01400=1040.303,84.994,410.568,169.774,38.664,157.276
C01401=1040.310,85.243,410.549,169.776,38.664,157.276
C01402=1040.316,85.492,410.530,169.777,38.665,157.276
C01403=1040.323,85.741,410.512,169.779,38.665,157.276
C01404=1040.329,85.991,410.493,169.782,38.666,157.277
C01405=1040.335,86.240,410.474,169.784,38.666,157.277
C01406=1040.341,86.489,410.455,169.786,38.667,157.277
C01407=1040.348,86.738,410.437,169.788,38.668,157.277
C01408=1040.354,86.987,410.418,169.790,38.668,157.277
C01409=1040.360,87.236,410.399,169.791,38.669,157.277
C01410=1040.366,87.486,410.380,169.793,38.670,157.278
C01411=1040.373,87.735,410.361,169.796,38.670,157.278
C01412=1040.379,87.984,410.343,169.798,38.671,157.278
C01413=1040.385,88.233,410.324,169.800,38.672,157.278
C01414=1040.392,88.483,410.304,169.802,38.672,157.278
C01415=1040.398,88.732,410.285,169.803,38.673,157.278
C01416=1040.405,88.981,410.266,169.805,38.673,157.279
C01417=1040.411,89.230,410.248,169.807,38.674,157.279
C01418=1040.417,89.480,410.229,169.810,38.674,157.279
C01419=1040.423,89.729,410.210,169.812,38.675,157.279
C01420=1040.430,89.978,410.191,169.814,38.676,157.279
C01421=1040.436,90.227,410.173,169.816,38.677,157.280
C01422=1040.442,90.476,410.153,169.817,38.677,157.280
C01423=1040.448,90.725,410.135,169.819,38.678,157.280
C01424=1040.454,90.974,410.115,169.822,38.679,157.280
C01425=1040.461,91.223,410.096,169.824,38.679,157.280
C01426=1040.466,91.473,410.077,169.826,38.680,157.280
C01427=1040.473,91.722,410.058,169.828,38.680,157.281
C01428=1040.479,91.972,410.039,169.829,38.682,157.281
C01429=1040.486,92.221,410.019,169.831,38.682,157.281
C01430=1040.492,92.470,410.000,169.833,38.683,157.281
C01431=1040.499,92.756,409.978,169.836,38.684,157.281
C01432=1040.506,93.041,409.956,169.838,38.684,157.282
C01433=1040.513,93.328,409.935,169.840,38.685,157.282
C01434=1040.520,93.613,409.912,169.842,38.686,157.282
C01435=1040.526,93.863,409.893,169.844,38.686,157.282
C01436=1040.532,94.112,409.874,169.846,38.687,157.282
C01437=1040.539,94.362,409.855,169.849,38.688,157.283
C01438=1040.545,94.611,409.835,169.851,38.689,157.283
C01439=1040.551,94.860,409.816,169.853,38.689,157.283
C01440=1040.557,95.109,409.797,169.855,38.690,157.283
C01441=1040.563,95.358,409.778,169.856,38.691,157.283
C01442=1040.569,95.607,409.758,169.858,38.691,157.283
C01443=1040.576,95.857,409.740,169.860,38.692,157.284
C01444=1040.582,96.105,409.720,169.863,38.692,157.284
C01445=1040.589,96.355,409.701,169.865,38.694,157.284
C01446=1040.594,96.605,409.682,169.867,38.694,157.284
C01447=1040.601,96.853,409.662,169.868,38.695,157.284
C01448=1040.607,97.103,409.643,169.870,38.695,157.284
C01449=1040.613,97.352,409.624,169.872,38.696,157.285
C01450=1040.619,97.600,409.604,169.875,38.697,157.285
C01451=1040.626,97.850,409.585,169.877,38.697,157.285
C01452=1040.632,98.099,409.565,169.879,38.698,157.285
C01453=1040.638,98.349,409.546,169.881,38.698,157.285
C01454=1040.644,98.598,409.528,169.882,38.700,157.286
C01455=1040.650,98.846,409.508,169.884,38.700,157.286
C01456=1040.657,99.096,409.489,169.886,38.701,157.286
C01457=1040.663,99.345,409.469,169.889,38.701,157.286
C01458=1040.670,99.594,409.450,169.891,38.702,157.286
C01459=1040.676,99.843,409.430,169.893,38.703,157.286
C01460=1040.682,100.092,409.411,169.895,38.703,157.287
C01461=1040.689,100.342,409.391,169.896,38.704,157.287
C01462=1040.694,100.591,409.372,169.898,38.705,157.287
C01463=1040.701,100.840,409.352,169.901,38.706,157.287
C01464=1040.707,101.089,409.333,169.903,38.706,157.287
C01465=1040.713,101.338,409.313,169.905,38.707,157.287
C01466=1040.719,101.588,409.294,169.907,38.708,157.288
C01467=1040.725,101.837,409.274,169.909,38.708,157.288
C01468=1040.731,102.086,409.255,169.910,38.709,157.288
C01469=1040.737,102.335,409.235,169.913,38.710,157.288
C01470=1040.743,102.584,409.215,169.915,38.711,157.288
C01471=1040.750,102.834,409.195,169.917,38.711,157.289
C01472=1040.756,103.082,409.176,169.919,38.712,157.289
C01473=1040.761,103.332,409.156,169.921,38.713,157.289
C01474=1040.768,103.580,409.137,169.922,38.713,157.289
C01475=1040.775,103.830,409.117,169.925,38.715,157.289
C01476=1040.780,104.079,409.097,169.927,38.715,157.290
C01477=1040.786,104.328,409.077,169.929,38.716,157.290
C01478=1040.792,104.577,409.057,169.931,38.717,157.290
C01479=1040.799,104.826,409.039,169.933,38.717,157.290
C01480=1040.805,105.076,409.018,169.935,38.718,157.290
C01481=1040.811,105.324,408.998,169.937,38.719,157.291
C01482=1040.817,105.574,408.979,169.939,38.719,157.291
C01483=1040.824,105.823,408.959,169.941,38.720,157.291
C01484=1040.830,106.072,408.939,169.943,38.721,157.291
C01485=1040.836,106.321,408.920,169.945,38.722,157.291
C01486=1040.842,106.570,408.900,169.947,38.722,157.292
C01487=1040.849,106.820,408.880,169.949,38.723,157.292
C01488=1040.854,107.069,408.861,169.951,38.724,157.292
C01489=1040.860,107.318,408.841,169.953,38.724,157.292
C01490=1040.867,107.567,408.820,169.955,38.725,157.292
C01491=1040.874,107.816,408.801,169.957,38.726,157.293
C01492=1040.879,108.065,408.782,169.959,38.727,157.293
C01493=1040.886,108.315,408.762,169.961,38.727,157.293
C01494=1040.892,108.564,408.742,169.964,38.728,157.293
C01495=1040.899,108.849,408.719,169.966,38.729,157.293
C01496=1040.906,109.135,408.696,169.968,38.729,157.293
C01497=1040.914,109.421,408.674,169.970,38.730,157.294
C01498=1040.921,109.708,408.651,169.972,38.731,157.294
C01499=1040.927,109.957,408.631,169.975,38.732,157.294
C01500=1040.933,110.205,408.611,169.977,38.733,157.294
C01501=1040.939,110.455,408.590,169.979,38.733,157.294
C01502=1040.945,110.704,408.571,169.981,38.734,157.295
C01503=1040.951,110.953,408.551,169.983,38.735,157.295
C01504=1040.958,111.203,408.531,169.985,38.735,157.295
C01505=1040.964,111.452,408.511,169.988,38.736,157.295
C01506=1040.970,111.700,408.491,169.989,38.737,157.295
C01507=1040.976,111.950,408.471,169.991,38.738,157.296
C01508=1040.982,112.199,408.451,169.993,38.739,157.296
C01509=1040.989,112.448,408.430,169.995,38.739,157.296
C01510=1040.995,112.697,408.410,169.997,38.740,157.296
C01511=1041.001,112.946,408.390,170.000,38.741,157.296
C01512=1041.008,113.195,408.370,170.002,38.741,157.297
C01513=1041.014,113.444,408.350,170.004,38.742,157.297
C01514=1041.020,113.693,408.330,170.005,38.743,157.297
C01515=1041.026,113.942,408.310,170.007,38.744,157.297
C01516=1041.032,114.191,408.290,170.009,38.745,157.297
C01517=1041.037,114.440,408.269,170.012,38.745,157.298
C01518=1041.044,114.690,408.249,170.014,38.746,157.298
C01519=1041.050,114.939,408.229,170.016,38.747,157.298
C01520=1041.056,115.188,408.209,170.018,38.748,157.298
C01521=1041.062,115.437,408.188,170.019,38.749,157.298
C01522=1041.068,115.686,408.168,170.022,38.750,157.299
C01523=1041.074,115.936,408.148,170.024,38.750,157.299
C01524=1041.080,116.185,408.128,170.026,38.751,157.299
C01525=1041.086,116.434,408.107,170.028,38.752,157.299
C01526=1041.092,116.683,408.087,170.030,38.753,157.300
C01527=1041.099,116.931,408.066,170.032,38.754,157.300
C01528=1041.104,117.180,408.046,170.034,38.755,157.300
C01529=1041.110,117.430,408.026,170.036,38.755,157.300
C01530=1041.116,117.679,408.006,170.038,38.756,157.300
C01531=1041.123,117.928,407.985,170.040,38.757,157.301
C01532=1041.128,118.177,407.965,170.042,38.758,157.301
C01533=1041.134,118.426,407.945,170.045,38.759,157.301
C01534=1041.141,118.675,407.924,170.047,38.760,157.301
C01535=1041.146,118.924,407.903,170.049,38.760,157.301
C01536=1041.153,119.174,407.883,170.051,38.761,157.302
C01537=1041.159,119.423,407.863,170.052,38.762,157.302
C01538=1041.166,119.672,407.843,170.054,38.762,157.302
C01539=1041.171,119.921,407.821,170.057,38.764,157.302
C01540=1041.178,120.170,407.801,170.059,38.764,157.302
C01541=1041.184,120.419,407.781,170.061,38.765,157.303
C01542=1041.189,120.668,407.760,170.063,38.766,157.303
C01543=1041.196,120.917,407.739,170.065,38.767,157.303
C01544=1041.202,121.166,407.719,170.068,38.767,157.303
C01545=1041.208,121.416,407.699,170.070,38.769,157.304
C01546=1041.214,121.664,407.679,170.071,38.769,157.304
C01547=1041.221,121.913,407.658,170.073,38.770,157.304
C01548=1041.227,122.162,407.638,170.075,38.771,157.304
C01549=1041.232,122.412,407.617,170.077,38.771,157.304
C01550=1041.238,122.661,407.597,170.080,38.772,157.305
C01551=1041.245,122.910,407.576,170.082,38.773,157.305
C01552=1041.251,123.159,407.555,170.084,38.774,157.305
C01553=1041.257,123.408,407.535,170.086,38.775,157.305
C01554=1041.264,123.656,407.514,170.088,38.776,157.305
C01555=1041.269,123.906,407.493,170.091,38.776,157.306
C01556=1041.275,124.155,407.473,170.093,38.777,157.306
C01557=1041.282,124.404,407.452,170.095,38.778,157.306
C01558=1041.288,124.654,407.431,170.096,38.779,157.306
C01559=1041.295,124.939,407.408,170.099,38.780,157.306
C01560=1041.302,125.225,407.384,170.102,38.781,157.307
C01561=1041.309,125.511,407.361,170.104,38.781,157.307
C01562=1041.316,125.797,407.337,170.106,38.782,157.307
C01563=1041.323,126.046,407.316,170.108,38.783,157.307
C01564=1041.329,126.295,407.295,170.110,38.784,157.308
C01565=1041.335,126.544,407.275,170.112,38.785,157.308
C01566=1041.341,126.792,407.254,170.115,38.786,157.308
C01567=1041.351,127.151,407.225,170.118,38.787,157.308
C01568=1041.359,127.509,407.194,170.121,38.788,157.309
C01569=1041.368,127.867,407.165,170.124,38.789,157.309
C01570=1041.377,128.225,407.135,170.127,38.790,157.309
C01571=1041.383,128.474,407.115,170.129,38.791,157.309
C01572=1041.390,128.723,407.094,170.131,38.792,157.310
C01573=1041.396,128.972,407.073,170.133,38.792,157.310
C01574=1041.402,129.221,407.052,170.135,38.793,157.310
C01575=1041.408,129.470,407.031,170.138,38.794,157.310
C01576=1041.415,129.719,407.010,170.140,38.794,157.310
C01577=1041.421,129.968,406.990,170.142,38.795,157.311
C01578=1041.427,130.217,406.968,170.144,38.796,157.311
C01579=1041.434,130.467,406.948,170.146,38.797,157.311
C01580=1041.440,130.715,406.927,170.149,38.798,157.311
C01581=1041.446,130.965,406.906,170.151,38.798,157.311
C01582=1041.453,131.214,406.885,170.153,38.799,157.312
C01583=1041.459,131.462,406.864,170.155,38.800,157.312
C01584=1041.465,131.712,406.844,170.157,38.801,157.312
C01585=1041.471,131.960,406.823,170.160,38.802,157.312
C01586=1041.477,132.210,406.801,170.162,38.803,157.313
C01587=1041.484,132.459,406.781,170.164,38.804,157.313
C01588=1041.489,132.708,406.759,170.166,38.804,157.313
C01589=1041.495,132.957,406.738,170.168,38.805,157.313
C01590=1041.502,133.206,406.717,170.169,38.806,157.313
C01591=1041.507,133.455,406.696,170.172,38.807,157.314
C01592=1041.514,133.704,406.674,170.174,38.808,157.314
C01593=1041.520,133.953,406.654,170.176,38.809,157.314
C01594=1041.526,134.202,406.633,170.178,38.810,157.314
C01595=1041.532,134.451,406.611,170.180,38.810,157.315
C01596=1041.539,134.700,406.590,170.183,38.811,157.315
C01597=1041.544,134.949,406.570,170.185,38.812,157.315
C01598=1041.550,135.198,406.548,170.187,38.813,157.315
C01599=1041.557,135.447,406.527,170.189,38.814,157.315
C01600=1041.563,135.696,406.506,170.191,38.815,157.316
C01601=1041.569,135.945,406.484,170.194,38.816,157.316
C01602=1041.575,136.195,406.463,170.196,38.816,157.316
C01603=1041.581,136.443,406.442,170.198,38.818,157.316
C01604=1041.587,136.692,406.421,170.200,38.818,157.317
C01605=1041.593,136.941,406.399,170.202,38.819,157.317
C01606=1041.600,137.190,406.378,170.205,38.820,157.317
C01607=1041.606,137.439,406.357,170.207,38.821,157.317
C01608=1041.612,137.689,406.336,170.209,38.822,157.318
C01609=1041.618,137.938,406.314,170.211,38.822,157.318
C01610=1041.625,138.187,406.293,170.213,38.824,157.318
C01611=1041.630,138.435,406.272,170.216,38.824,157.318
C01612=1041.636,138.684,406.250,170.218,38.825,157.318
C01613=1041.643,138.934,406.229,170.220,38.826,157.319
C01614=1041.649,139.182,406.208,170.222,38.827,157.319
C01615=1041.655,139.431,406.186,170.224,38.828,157.319
C01616=1041.661,139.680,406.165,170.227,38.829,157.319
C01617=1041.667,139.929,406.143,170.229,38.830,157.320
C01618=1041.673,140.178,406.122,170.231,38.831,157.320
C01619=1041.679,140.391,406.104,170.232,38.831,157.320
C01620=1041.683,140.604,406.085,170.234,38.832,157.320
C01621=1041.689,140.818,406.067,170.237,38.833,157.320
C01622=1041.694,141.030,406.049,170.239,38.833,157.321
C01623=1041.699,141.243,406.031,170.240,38.835,157.321
C01624=1041.704,141.456,406.011,170.242,38.835,157.321
C01625=1041.710,141.669,405.993,170.244,38.836,157.321
C01626=1041.715,141.881,405.975,170.245,38.837,157.321
C01627=1041.721,142.130,405.954,170.248,38.838,157.322
C01628=1041.727,142.380,405.932,170.250,38.839,157.322
C01629=1041.733,142.629,405.910,170.252,38.840,157.322
C01630=1041.739,142.878,405.889,170.254,38.841,157.322
C01631=1041.745,143.126,405.868,170.256,38.841,157.323
C01632=1041.751,143.376,405.846,170.259,38.842,157.323
C01633=1041.758,143.624,405.824,170.261,38.844,157.323
C01634=1041.764,143.873,405.802,170.263,38.844,157.323
C01635=1041.770,144.123,405.780,170.265,38.845,157.324
C01636=1041.775,144.371,405.759,170.268,38.846,157.324
C01637=1041.782,144.620,405.737,170.270,38.847,157.324
C01638=1041.788,144.870,405.716,170.272,38.848,157.324
C01639=1041.794,145.119,405.694,170.274,38.849,157.325
C01640=1041.800,145.367,405.672,170.276,38.850,157.325
C01641=1041.807,145.617,405.650,170.279,38.851,157.325
C01642=1041.813,145.865,405.629,170.282,38.852,157.325
C01643=1041.819,146.114,405.608,170.284,38.852,157.325
C01644=1041.825,146.363,405.586,170.286,38.853,157.326
C01645=1041.831,146.612,405.565,170.289,38.855,157.326
C01646=1041.838,146.861,405.542,170.291,38.855,157.326
C01647=1041.844,147.110,405.521,170.293,38.856,157.326
C01648=1041.850,147.359,405.499,170.295,38.857,157.327
C01649=1041.856,147.609,405.477,170.297,38.858,157.327
C01650=1041.861,147.857,405.455,170.300,38.859,157.327
C01651=1041.868,148.106,405.433,170.302,38.860,157.327
C01652=1041.874,148.355,405.411,170.304,38.861,157.328
C01653=1041.880,148.604,405.389,170.306,38.862,157.328
C01654=1041.886,148.853,405.367,170.308,38.863,157.328
C01655=1041.893,149.102,405.346,170.311,38.864,157.328
C01656=1041.899,149.351,405.323,170.313,38.865,157.329
C01657=1041.905,149.600,405.301,170.315,38.866,157.329
C01658=1041.910,149.849,405.280,170.317,38.867,157.329
C01659=1041.917,150.097,405.258,170.320,38.868,157.329
C01660=1041.923,150.347,405.236,170.322,38.869,157.330
C01661=1041.929,150.596,405.214,170.324,38.870,157.330
C01662=1041.935,150.845,405.191,170.326,38.871,157.330
C01663=1041.941,151.094,405.170,170.328,38.872,157.330
C01664=1041.947,151.342,405.147,170.331,38.873,157.331
C01665=1041.953,151.592,405.126,170.333,38.874,157.331
C01666=1041.960,151.841,405.104,170.335,38.875,157.331
C01667=1041.965,152.090,405.081,170.338,38.876,157.332
C01668=1041.971,152.339,405.060,170.341,38.877,157.332
C01669=1041.978,152.588,405.037,170.343,38.878,157.332
C01670=1041.984,152.837,405.016,170.345,38.879,157.332
C01671=1041.990,153.085,404.994,170.347,38.880,157.333
C01672=1041.995,153.334,404.971,170.350,38.881,157.333
C01673=1042.002,153.583,404.949,170.352,38.882,157.333
C01674=1042.008,153.832,404.927,170.354,38.883,157.333
C01675=1042.014,154.081,404.905,170.356,38.884,157.334
C01676=1042.020,154.330,404.883,170.358,38.884,157.334
C01677=1042.026,154.579,404.860,170.361,38.886,157.334
C01678=1042.033,154.828,404.839,170.363,38.887,157.334
C01679=1042.038,155.077,404.816,170.365,38.888,157.335
C01680=1042.045,155.325,404.793,170.367,38.889,157.335
C01681=1042.051,155.575,404.772,170.370,38.890,157.335
C01682=1042.057,155.823,404.749,170.373,38.891,157.336
C01683=1042.063,156.073,404.727,170.375,38.892,157.336
C01684=1042.069,156.321,404.705,170.377,38.893,157.336
C01685=1042.075,156.570,404.682,170.380,38.894,157.336
C01686=1042.081,156.819,404.660,170.382,38.895,157.337
C01687=1042.089,157.105,404.634,170.384,38.896,157.337
C01688=1042.095,157.390,404.609,170.387,38.897,157.337
C01689=1042.102,157.675,404.583,170.390,38.898,157.337
C01690=1042.109,157.961,404.557,170.393,38.899,157.338
C01691=1042.116,158.209,404.535,170.395,38.900,157.338
C01692=1042.122,158.459,404.513,170.397,38.902,157.338
C01693=1042.127,158.708,404.490,170.400,38.903,157.339
C01694=1042.134,158.956,404.468,170.402,38.904,157.339
C01695=1042.140,159.205,404.445,170.404,38.905,157.339
C01696=1042.146,159.454,404.423,170.406,38.906,157.339
C01697=1042.152,159.703,404.401,170.409,38.907,157.340
C01698=1042.158,159.952,404.378,170.411,38.908,157.340
C01699=1042.165,160.200,404.356,170.414,38.909,157.340
C01700=1042.170,160.450,404.334,170.416,38.910,157.340
C01701=1042.176,160.699,404.311,170.419,38.911,157.341
C01702=1042.182,160.947,404.288,170.421,38.912,157.341
C01703=1042.188,161.196,404.265,170.423,38.913,157.341
C01704=1042.194,161.445,404.242,170.425,38.915,157.342
C01705=1042.199,161.694,404.219,170.428,38.916,157.342
C01706=1042.205,161.943,404.197,170.430,38.917,157.342
C01707=1042.212,162.191,404.174,170.432,38.918,157.343
C01708=1042.217,162.440,404.151,170.434,38.919,157.343
C01709=1042.223,162.691,404.129,170.437,38.921,157.343
C01710=1042.229,162.940,404.106,170.439,38.922,157.343
C01711=1042.235,163.188,404.083,170.442,38.923,157.344
C01712=1042.241,163.437,404.060,170.444,38.924,157.344
C01713=1042.247,163.686,404.037,170.447,38.925,157.344
C01714=1042.253,163.935,404.015,170.449,38.926,157.345
C01715=1042.258,164.184,403.992,170.451,38.927,157.345
C01716=1042.265,164.432,403.969,170.454,38.929,157.345
C01717=1042.271,164.681,403.946,170.456,38.930,157.346
C01718=1042.276,164.930,403.923,170.458,38.931,157.346
C01719=1042.282,165.179,403.900,170.460,38.932,157.346
C01720=1042.288,165.428,403.877,170.464,38.933,157.346
C01721=1042.295,165.676,403.854,170.466,38.935,157.347
C01722=1042.300,165.925,403.831,170.468,38.936,157.347
C01723=1042.307,166.174,403.808,170.470,38.937,157.347
C01724=1042.312,166.423,403.785,170.473,38.938,157.348
C01725=1042.318,166.672,403.762,170.475,38.939,157.348
C01726=1042.325,166.921,403.740,170.477,38.940,157.348
C01727=1042.330,167.170,403.717,170.481,38.942,157.349
C01728=1042.336,167.418,403.694,170.483,38.943,157.349
C01729=1042.342,167.667,403.671,170.485,38.944,157.349
C01730=1042.348,167.917,403.648,170.487,38.945,157.349
C01731=1042.354,168.165,403.624,170.490,38.946,157.350
C01732=1042.361,168.414,403.602,170.492,38.947,157.350
C01733=1042.366,168.663,403.579,170.494,38.949,157.350
C01734=1042.372,168.912,403.556,170.497,38.950,157.351
C01735=1042.378,169.161,403.533,170.500,38.951,157.351
C01736=1042.384,169.410,403.510,170.502,38.952,157.351
C01737=1042.390,169.658,403.486,170.504,38.954,157.352
C01738=1042.397,169.907,403.464,170.506,38.955,157.352
C01739=1042.402,170.156,403.441,170.509,38.956,157.352
C01740=1042.408,170.405,403.418,170.512,38.957,157.352
C01741=1042.415,170.654,403.394,170.514,38.958,157.353
C01742=1042.420,170.903,403.371,170.517,38.959,157.353
C01743=1042.426,171.152,403.348,170.519,38.960,157.353
C01744=1042.433,171.400,403.325,170.521,38.961,157.354
C01745=1042.439,171.649,403.301,170.524,38.962,157.354
C01746=1042.445,171.898,403.278,170.527,38.964,157.354
C01747=1042.451,172.147,403.255,170.529,38.965,157.355
C01748=1042.457,172.396,403.233,170.531,38.966,157.355
C01749=1042.463,172.645,403.208,170.533,38.967,157.355
C01750=1042.469,172.894,403.186,170.537,38.968,157.355
C01751=1042.477,173.178,403.159,170.539,38.970,157.356
C01752=1042.483,173.463,403.133,170.542,38.971,157.356
C01753=1042.490,173.748,403.106,170.545,38.972,157.356
C01754=1042.497,174.033,403.079,170.548,38.974,157.357
C01755=1042.503,174.282,403.056,170.550,38.975,157.357
C01756=1042.509,174.530,403.032,170.553,38.976,157.357
C01757=1042.515,174.780,403.009,170.555,38.977,157.358
C01758=1042.522,175.028,402.987,170.558,38.978,157.358
C01759=1042.528,175.277,402.963,170.560,38.980,157.358
C01760=1042.534,175.526,402.940,170.563,38.981,157.359
C01761=1042.540,175.774,402.916,170.565,38.982,157.359
C01762=1042.546,176.023,402.893,170.568,38.983,157.359
C01763=1042.553,176.272,402.869,170.570,38.985,157.360
C01764=1042.558,176.521,402.846,170.573,38.986,157.360
C01765=1042.564,176.770,402.823,170.575,38.987,157.360
C01766=1042.572,177.019,402.800,170.578,38.988,157.360
C01767=1042.577,177.268,402.777,170.581,38.990,157.361
C01768=1042.584,177.517,402.753,170.583,38.991,157.361
C01769=1042.590,177.765,402.729,170.585,38.992,157.361
C01770=1042.596,178.014,402.706,170.588,38.993,157.362
C01771=1042.602,178.263,402.682,170.591,38.994,157.362
C01772=1042.608,178.512,402.659,170.593,38.995,157.362
C01773=1042.615,178.761,402.635,170.596,38.997,157.363
C01774=1042.620,179.010,402.612,170.599,38.998,157.363
C01775=1042.626,179.258,402.589,170.601,38.999,157.363
C01776=1042.634,179.507,402.566,170.603,39.000,157.364
C01777=1042.640,179.755,402.542,170.606,39.001,157.364
C01778=1042.646,180.004,402.518,170.609,39.002,157.364
C01779=1042.652,180.253,402.495,170.611,39.004,157.365
C01780=1042.659,180.502,402.471,170.614,39.005,157.365
C01781=1042.664,180.751,402.448,170.617,39.006,157.365
C01782=1042.671,181.000,402.424,170.619,39.007,157.365
C01783=1042.677,181.248,402.401,170.621,39.008,157.366
C01784=1042.683,181.498,402.377,170.624,39.009,157.366
C01785=1042.689,181.746,402.354,170.627,39.011,157.366
C01786=1042.696,181.995,402.330,170.629,39.012,157.367
C01787=1042.702,182.244,402.307,170.632,39.013,157.367
C01788=1042.708,182.493,402.283,170.634,39.014,157.367
C01789=1042.715,182.741,402.260,170.637,39.015,157.368
C01790=1042.721,182.991,402.236,170.640,39.017,157.368
C01791=1042.727,183.239,402.213,170.642,39.018,157.368
C01792=1042.734,183.488,402.189,170.645,39.019,157.369
C01793=1042.740,183.736,402.165,170.648,39.020,157.369
C01794=1042.746,183.986,402.140,170.650,39.022,157.369
C01795=1042.752,184.234,402.117,170.653,39.023,157.370
C01796=1042.758,184.484,402.093,170.656,39.025,157.370
C01797=1042.764,184.732,402.069,170.658,39.026,157.370
C01798=1042.769,184.981,402.045,170.661,39.028,157.371
C01799=1042.776,185.230,402.021,170.663,39.029,157.371
C01800=1042.781,185.478,401.997,170.666,39.030,157.371
C01801=1042.788,185.727,401.973,170.669,39.032,157.372
C01802=1042.793,185.976,401.948,170.671,39.033,157.372
C01803=1042.800,186.225,401.924,170.674,39.034,157.372
C01804=1042.805,186.473,401.900,170.677,39.036,157.373
C01805=1042.811,186.722,401.876,170.679,39.037,157.373
C01806=1042.817,186.971,401.852,170.681,39.039,157.374
C01807=1042.823,187.220,401.828,170.684,39.040,157.374
C01808=1042.829,187.468,401.803,170.687,39.042,157.374
C01809=1042.835,187.717,401.779,170.689,39.043,157.375
C01810=1042.841,187.966,401.755,170.693,39.044,157.375
C01811=1042.847,188.215,401.731,170.695,39.046,157.375
C01812=1042.853,188.464,401.707,170.697,39.047,157.376
C01813=1042.859,188.713,401.683,170.701,39.049,157.376
C01814=1042.865,188.961,401.659,170.703,39.050,157.376
